LIN {X 0,Y 300.537,Z 1135.109,A -85,B 0,C 180,E1 14462.884,E2 14462.884} C_VEL
LIN {X 0,Y 304.265,Z 1129.427,A -85,B 0,C 180,E1 14457.835,E2 14457.835} C_VEL
LIN {X 0,Y 309.402,Z 1122.153,A -85,B 0,C 180,E1 14453.053,E2 14453.053} C_VEL
LIN {X 0,Y 314.973,Z 1114.845,A -85,B 0,C 180,E1 14449.161,E2 14449.161} C_VEL
LIN {X 0,Y 322.841,Z 1104.94,A -85,B 0,C 180,E1 14444.828,E2 14444.828} C_VEL
LIN {X 0,Y 331.827,Z 1093.472,A -85,B 0,C 180,E1 14440.835,E2 14440.835} C_VEL
LIN {X 0,Y 340.361,Z 1082.576,A -85,B 0,C 180,E1 14437.666,E2 14437.666} C_VEL
LIN {X 0,Y 350.994,Z 1068.769,A -85,B 0,C 180,E1 14434.299,E2 14434.299} C_VEL
LIN {X 0,Y 362.344,Z 1053.189,A -85,B 0,C 180,E1 14431.194,E2 14431.194} C_VEL
LIN {X 0,Y 369.861,Z 1042.527,A -85,B 0,C 180,E1 14429.373,E2 14429.373} C_VEL
LIN {X 0,Y 372.476,Z 1037.928,A -85,B 0,C 180,E1 14428.507,E2 14428.507} C_VEL
LIN {X 0,Y 377.031,Z 1026.802,A -85,B 0,C 180,E1 14426.039,E2 14426.039} C_VEL
LIN {X 0,Y 379.887,Z 1021.809,A -85,B 0,C 180,E1 14425.24,E2 14425.24} C_VEL
LIN {X 0,Y 392.376,Z 1001.673,A -85,B 0,C 180,E1 14422.92,E2 14422.92} C_VEL
LIN {X 0,Y 402.293,Z 984.331,A -85,B 0,C 180,E1 14421.248,E2 14421.248} C_VEL
LIN {X 0,Y 411.726,Z 966.45,A -85,B 0,C 180,E1 14419.775,E2 14419.775} C_VEL
LIN {X 0,Y 422.966,Z 942.726,A -85,B 0,C 180,E1 14418.141,E2 14418.141} C_VEL
LIN {X 0,Y 431.437,Z 922.389,A -85,B 0,C 180,E1 14416.979,E2 14416.979} C_VEL
LIN {X 0,Y 438.973,Z 902.071,A -85,B 0,C 180,E1 14415.999,E2 14415.999} C_VEL
LIN {X 0,Y 446.899,Z 877.548,A -85,B 0,C 180,E1 14415.019,E2 14415.019} C_VEL
LIN {X 0,Y 453.336,Z 852.946,A -85,B 0,C 180,E1 14414.24,E2 14414.24} C_VEL
LIN {X 0,Y 457.711,Z 832.707,A -85,B 0,C 180,E1 14413.717,E2 14413.717} C_VEL
LIN {X 0,Y 461.683,Z 809.62,A -85,B 0,C 180,E1 14413.245,E2 14413.245} C_VEL
LIN {X 0,Y 465.62,Z 774.989,A -85,B 0,C 180,E1 14412.698,E2 14412.698} C_VEL
LIN {X 0,Y 486.7,Z 556.586,A -85,B 0,C 180,E1 14409.493,E2 14409.493} C_VEL
LIN {X 0,Y 483.697,Z 550.634,A -85,B 0,C 180,E1 14407.185,E2 14407.185} C_VEL
LIN {X 0,Y 481.77,Z 547.068,A -85,B 0,C 180,E1 14405.359,E2 14405.359} C_VEL
LIN {X 0,Y 479.853,Z 543.385,A -85,B 0,C 180,E1 14402.867,E2 14402.867} C_VEL
LIN {X 0,Y 478.312,Z 540.425,A -85,B 0,C 180,E1 14398.443,E2 14398.443} C_VEL
LIN {X 0,Y 478.408,Z 540.862,A -85,B 0,C 180,E1 14396.285,E2 14396.285} C_VEL
LIN {X 0,Y 480.24,Z 544.178,A -85,B 0,C 180,E1 14392.162,E2 14392.162} C_VEL
LIN {X 0,Y 482.636,Z 548.887,A -85,B 0,C 180,E1 14389.375,E2 14389.375} C_VEL
LIN {X 0,Y 485.723,Z 554.856,A -85,B 0,C 180,E1 14386.822,E2 14386.822} C_VEL
LIN {X 0,Y 487.472,Z 558.564,A -85,B 0,C 180,E1 14385.592,E2 14385.592} C_VEL
LIN {X 0,Y 466.374,Z 778.807,A -85,B 0,C 180,E1 14382.251,E2 14382.251} C_VEL
LIN {X 0,Y 462.156,Z 819.105,A -85,B 0,C 180,E1 14381.613,E2 14381.613} C_VEL
LIN {X 0,Y 457.701,Z 845.254,A -85,B 0,C 180,E1 14381.12,E2 14381.12} C_VEL
LIN {X 0,Y 452.901,Z 867.044,A -85,B 0,C 180,E1 14380.637,E2 14380.637} C_VEL
LIN {X 0,Y 446.872,Z 889.838,A -85,B 0,C 180,E1 14380.007,E2 14380.007} C_VEL
LIN {X 0,Y 438.226,Z 917.079,A -85,B 0,C 180,E1 14379.046,E2 14379.046} C_VEL
LIN {X 0,Y 430.44,Z 938.212,A -85,B 0,C 180,E1 14378.123,E2 14378.123} C_VEL
LIN {X 0,Y 422.65,Z 957.244,A -85,B 0,C 180,E1 14377.137,E2 14377.137} C_VEL
LIN {X 0,Y 413.874,Z 976.767,A -85,B 0,C 180,E1 14375.95,E2 14375.95} C_VEL
LIN {X 0,Y 402.017,Z 1000.765,A -85,B 0,C 180,E1 14374.202,E2 14374.202} C_VEL
LIN {X 0,Y 390.581,Z 1021.665,A -85,B 0,C 180,E1 14372.342,E2 14372.342} C_VEL
LIN {X 0,Y 380.886,Z 1038.311,A -85,B 0,C 180,E1 14370.6,E2 14370.6} C_VEL
LIN {X 0,Y 370.782,Z 1054.723,A -85,B 0,C 180,E1 14368.607,E2 14368.607} C_VEL
LIN {X 0,Y 358.615,Z 1073.631,A -85,B 0,C 180,E1 14365.901,E2 14365.901} C_VEL
LIN {X 0,Y 346.466,Z 1091.434,A -85,B 0,C 180,E1 14362.797,E2 14362.797} C_VEL
LIN {X 0,Y 336.904,Z 1105.17,A -85,B 0,C 180,E1 14359.968,E2 14359.968} C_VEL
LIN {X 0,Y 327.706,Z 1118.263,A -85,B 0,C 180,E1 14356.82,E2 14356.82} C_VEL
LIN {X 0,Y 317.452,Z 1133.02,A -85,B 0,C 180,E1 14352.623,E2 14352.623} C_VEL
LIN {X 0,Y 308.488,Z 1146.151,A -85,B 0,C 180,E1 14348.012,E2 14348.012} C_VEL
LIN {X 0,Y 302.311,Z 1155.803,A -85,B 0,C 180,E1 14343.983,E2 14343.983} C_VEL
LIN {X 0,Y 297.196,Z 1164.602,A -85,B 0,C 180,E1 14339.64,E2 14339.64} C_VEL
LIN {X 0,Y 292.558,Z 1173.912,A -85,B 0,C 180,E1 14333.998,E2 14333.998} C_VEL
LIN {X 0,Y 290.123,Z 1180.103,A -85,B 0,C 180,E1 14329.208,E2 14329.208} C_VEL
LIN {X 0,Y 288.961,Z 1184.384,A -85,B 0,C 180,E1 14325.041,E2 14325.041} C_VEL
LIN {X 0,Y 288.442,Z 1187.555,A -85,B 0,C 180,E1 14320.991,E2 14320.991} C_VEL
LIN {X 0,Y 288.367,Z 1189.644,A -85,B 0,C 180,E1 14317.171,E2 14317.171} C_VEL
LIN {X 0,Y 288.427,Z 1190.814,A -85,B 0,C 180,E1 14313.379,E2 14313.379} C_VEL
LIN {X 0,Y 288.471,Z 1191.053,A -85,B 0,C 180,E1 14309.603,E2 14309.603} C_VEL
LIN {X 0,Y 288.431,Z 1190.344,A -85,B 0,C 180,E1 14305.825,E2 14305.825} C_VEL
LIN {X 0,Y 288.4,Z 1188.559,A -85,B 0,C 180,E1 14301.828,E2 14301.828} C_VEL
LIN {X 0,Y 288.599,Z 1185.626,A -85,B 0,C 180,E1 14297.697,E2 14297.697} C_VEL
LIN {X 0,Y 289.271,Z 1181.807,A -85,B 0,C 180,E1 14293.742,E2 14293.742} C_VEL
LIN {X 0,Y 290.606,Z 1176.811,A -85,B 0,C 180,E1 14289.666,E2 14289.666} C_VEL
LIN {X 0,Y 292.787,Z 1170.706,A -85,B 0,C 180,E1 14285.593,E2 14285.593} C_VEL
LIN {X 0,Y 295.918,Z 1163.458,A -85,B 0,C 180,E1 14281.549,E2 14281.549} C_VEL
LIN {X 0,Y 301.052,Z 1153.247,A -85,B 0,C 180,E1 14276.77,E2 14276.77} C_VEL
LIN {X 0,Y 307.763,Z 1141.001,A -85,B 0,C 180,E1 14272.119,E2 14272.119} C_VEL
LIN {X 0,Y 314.195,Z 1129.927,A -85,B 0,C 180,E1 14268.554,E2 14268.554} C_VEL
LIN {X 0,Y 321.498,Z 1117.681,A -85,B 0,C 180,E1 14265.162,E2 14265.162} C_VEL
LIN {X 0,Y 331.215,Z 1101.671,A -85,B 0,C 180,E1 14261.386,E2 14261.386} C_VEL
LIN {X 0,Y 341.43,Z 1084.347,A -85,B 0,C 180,E1 14258.024,E2 14258.024} C_VEL
LIN {X 0,Y 350.126,Z 1069.288,A -85,B 0,C 180,E1 14255.524,E2 14255.524} C_VEL
LIN {X 0,Y 359.111,Z 1053.183,A -85,B 0,C 180,E1 14253.21,E2 14253.21} C_VEL
LIN {X 0,Y 370.02,Z 1032.783,A -85,B 0,C 180,E1 14250.712,E2 14250.712} C_VEL
LIN {X 0,Y 380.326,Z 1011.808,A -85,B 0,C 180,E1 14248.587,E2 14248.587} C_VEL
LIN {X 0,Y 388.737,Z 993.522,A -85,B 0,C 180,E1 14246.999,E2 14246.999} C_VEL
LIN {X 0,Y 396.864,Z 974.565,A -85,B 0,C 180,E1 14245.586,E2 14245.586} C_VEL
LIN {X 0,Y 406.006,Z 951.26,A -85,B 0,C 180,E1 14244.107,E2 14244.107} C_VEL
LIN {X 0,Y 414.426,Z 926.626,A -85,B 0,C 180,E1 14242.835,E2 14242.835} C_VEL
LIN {X 0,Y 420.697,Z 905.998,A -85,B 0,C 180,E1 14241.953,E2 14241.953} C_VEL
LIN {X 0,Y 426.292,Z 884.993,A -85,B 0,C 180,E1 14241.2,E2 14241.2} C_VEL
LIN {X 0,Y 432.216,Z 858.983,A -85,B 0,C 180,E1 14240.452,E2 14240.452} C_VEL
LIN {X 0,Y 436.823,Z 831.955,A -85,B 0,C 180,E1 14239.859,E2 14239.859} C_VEL
LIN {X 0,Y 439.519,Z 809.536,A -85,B 0,C 180,E1 14239.442,E2 14239.442} C_VEL
LIN {X 0,Y 456.799,Z 596.987,A -85,B 0,C 180,E1 14236.09,E2 14236.09} C_VEL
LIN {X 0,Y 461.245,Z 542.225,A -85,B 0,C 180,E1 14235.207,E2 14235.207} C_VEL
LIN {X 0,Y 455.004,Z 530.522,A -85,B 0,C 180,E1 14232.598,E2 14232.598} C_VEL
LIN {X 0,Y 449.602,Z 520.756,A -85,B 0,C 180,E1 14229.99,E2 14229.99} C_VEL
LIN {X 0,Y 444.95,Z 512.775,A -85,B 0,C 180,E1 14227.359,E2 14227.359} C_VEL
LIN {X 0,Y 441.664,Z 507.167,A -85,B 0,C 180,E1 14225.131,E2 14225.131} C_VEL
LIN {X 0,Y 438.229,Z 501.32,A -85,B 0,C 180,E1 14222.223,E2 14222.223} C_VEL
LIN {X 0,Y 435.396,Z 496.62,A -85,B 0,C 180,E1 14218.816,E2 14218.816} C_VEL
LIN {X 0,Y 433.481,Z 493.881,A -85,B 0,C 180,E1 14213.909,E2 14213.909} C_VEL
LIN {X 0,Y 433.569,Z 494.107,A -85,B 0,C 180,E1 14211.111,E2 14211.111} C_VEL
LIN {X 0,Y 435.686,Z 496.998,A -85,B 0,C 180,E1 14206.394,E2 14206.394} C_VEL
LIN {X 0,Y 438.693,Z 502.126,A -85,B 0,C 180,E1 14202.969,E2 14202.969} C_VEL
LIN {X 0,Y 442.524,Z 508.361,A -85,B 0,C 180,E1 14199.913,E2 14199.913} C_VEL
LIN {X 0,Y 446.976,Z 516.099,A -85,B 0,C 180,E1 14197.093,E2 14197.093} C_VEL
LIN {X 0,Y 451.772,Z 524.554,A -85,B 0,C 180,E1 14194.572,E2 14194.572} C_VEL
LIN {X 0,Y 457.944,Z 536.068,A -85,B 0,C 180,E1 14191.789,E2 14191.789} C_VEL
LIN {X 0,Y 458.382,Z 537.284,A -85,B 0,C 180,E1 14191.59,E2 14191.59} C_VEL
LIN {X 0,Y 439.079,Z 769.572,A -85,B 0,C 180,E1 14188.029,E2 14188.029} C_VEL
LIN {X 0,Y 435.642,Z 805.367,A -85,B 0,C 180,E1 14187.439,E2 14187.439} C_VEL
LIN {X 0,Y 431.934,Z 829.629,A -85,B 0,C 180,E1 14186.906,E2 14186.906} C_VEL
LIN {X 0,Y 427.887,Z 850.615,A -85,B 0,C 180,E1 14186.314,E2 14186.314} C_VEL
LIN {X 0,Y 422.274,Z 874.564,A -85,B 0,C 180,E1 14185.486,E2 14185.486} C_VEL
LIN {X 0,Y 415.381,Z 898.542,A -85,B 0,C 180,E1 14184.448,E2 14184.448} C_VEL
LIN {X 0,Y 408.612,Z 919.046,A -85,B 0,C 180,E1 14183.379,E2 14183.379} C_VEL
LIN {X 0,Y 400.988,Z 939.639,A -85,B 0,C 180,E1 14182.11,E2 14182.11} C_VEL
LIN {X 0,Y 390.967,Z 963.549,A -85,B 0,C 180,E1 14180.334,E2 14180.334} C_VEL
LIN {X 0,Y 382.521,Z 981.74,A -85,B 0,C 180,E1 14178.719,E2 14178.719} C_VEL
LIN {X 0,Y 374.05,Z 998.65,A -85,B 0,C 180,E1 14176.977,E2 14176.977} C_VEL
LIN {X 0,Y 363.351,Z 1018.538,A -85,B 0,C 180,E1 14174.563,E2 14174.563} C_VEL
LIN {X 0,Y 352.953,Z 1036.284,A -85,B 0,C 180,E1 14171.955,E2 14171.955} C_VEL
LIN {X 0,Y 344.235,Z 1050.501,A -85,B 0,C 180,E1 14169.502,E2 14169.502} C_VEL
LIN {X 0,Y 334.277,Z 1066.205,A -85,B 0,C 180,E1 14166.316,E2 14166.316} C_VEL
LIN {X 0,Y 324.82,Z 1080.383,A -85,B 0,C 180,E1 14162.803,E2 14162.803} C_VEL
LIN {X 0,Y 317.181,Z 1091.77,A -85,B 0,C 180,E1 14159.456,E2 14159.456} C_VEL
LIN {X 0,Y 309.26,Z 1103.755,A -85,B 0,C 180,E1 14155.262,E2 14155.262} C_VEL
LIN {X 0,Y 302.465,Z 1114.131,A -85,B 0,C 180,E1 14150.714,E2 14150.714} C_VEL
LIN {X 0,Y 297.915,Z 1121.561,A -85,B 0,C 180,E1 14146.776,E2 14146.776} C_VEL
LIN {X 0,Y 293.861,Z 1128.975,A -85,B 0,C 180,E1 14141.979,E2 14141.979} C_VEL
LIN {X 0,Y 291.048,Z 1134.872,A -85,B 0,C 180,E1 14136.906,E2 14136.906} C_VEL
LIN {X 0,Y 289.685,Z 1138.521,A -85,B 0,C 180,E1 14132.77,E2 14132.77} C_VEL
LIN {X 0,Y 289.008,Z 1141.071,A -85,B 0,C 180,E1 14128.81,E2 14128.81} C_VEL
LIN {X 0,Y 288.706,Z 1142.744,A -85,B 0,C 180,E1 14124.834,E2 14124.834} C_VEL
LIN {X 0,Y 288.659,Z 1143.577,A -85,B 0,C 180,E1 14120.63,E2 14120.63} C_VEL
LIN {X 0,Y 288.869,Z 1143.374,A -85,B 0,C 180,E1 14115.742,E2 14115.742} C_VEL
LIN {X 0,Y 289.497,Z 1141.838,A -85,B 0,C 180,E1 14111.055,E2 14111.055} C_VEL
LIN {X 0,Y 290.733,Z 1139.376,A -85,B 0,C 180,E1 14106.703,E2 14106.703} C_VEL
LIN {X 0,Y 292.756,Z 1136.021,A -85,B 0,C 180,E1 14102.544,E2 14102.544} C_VEL
LIN {X 0,Y 296.29,Z 1130.917,A -85,B 0,C 180,E1 14097.779,E2 14097.779} C_VEL
LIN {X 0,Y 301.799,Z 1123.582,A -85,B 0,C 180,E1 14092.669,E2 14092.669} C_VEL
LIN {X 0,Y 307.578,Z 1116.356,A -85,B 0,C 180,E1 14088.673,E2 14088.673} C_VEL
LIN {X 0,Y 314.486,Z 1107.977,A -85,B 0,C 180,E1 14084.847,E2 14084.847} C_VEL
LIN {X 0,Y 324.399,Z 1096.058,A -85,B 0,C 180,E1 14080.421,E2 14080.421} C_VEL
LIN {X 0,Y 333.918,Z 1084.361,A -85,B 0,C 180,E1 14076.919,E2 14076.919} C_VEL
LIN {X 0,Y 343.428,Z 1072.444,A -85,B 0,C 180,E1 14073.927,E2 14073.927} C_VEL
LIN {X 0,Y 354.974,Z 1057.507,A -85,B 0,C 180,E1 14070.785,E2 14070.785} C_VEL
LIN {X 0,Y 366.845,Z 1040.993,A -85,B 0,C 180,E1 14067.957,E2 14067.957} C_VEL
LIN {X 0,Y 376.707,Z 1026.562,A -85,B 0,C 180,E1 14065.871,E2 14065.871} C_VEL
LIN {X 0,Y 379.887,Z 1021.809,A -85,B 0,C 180,E1 14065.24,E2 14065.24} C_VEL
LIN {X 0,Y 382.759,Z 1016.786,A -85,B 0,C 180,E1 14064.46,E2 14064.46} C_VEL
LIN {X 0,Y 387.816,Z 1004.51,A -85,B 0,C 180,E1 14062.214,E2 14062.214} C_VEL
LIN {X 0,Y 390.69,Z 999.056,A -85,B 0,C 180,E1 14061.518,E2 14061.518} C_VEL
LIN {X 0,Y 402,Z 979.461,A -85,B 0,C 180,E1 14059.711,E2 14059.711} C_VEL
LIN {X 0,Y 413.33,Z 957.464,A -85,B 0,C 180,E1 14058.038,E2 14058.038} C_VEL
LIN {X 0,Y 422.043,Z 938.688,A -85,B 0,C 180,E1 14056.841,E2 14056.841} C_VEL
LIN {X 0,Y 429.75,Z 920.272,A -85,B 0,C 180,E1 14055.835,E2 14055.835} C_VEL
LIN {X 0,Y 438.408,Z 896.971,A -85,B 0,C 180,E1 14054.761,E2 14054.761} C_VEL
LIN {X 0,Y 446.121,Z 871.943,A -85,B 0,C 180,E1 14053.83,E2 14053.83} C_VEL
LIN {X 0,Y 451.666,Z 850.593,A -85,B 0,C 180,E1 14053.189,E2 14053.189} C_VEL
LIN {X 0,Y 456.216,Z 829.368,A -85,B 0,C 180,E1 14052.672,E2 14052.672} C_VEL
LIN {X 0,Y 460.774,Z 800.806,A -85,B 0,C 180,E1 14052.134,E2 14052.134} C_VEL
LIN {X 0,Y 467.223,Z 736.827,A -85,B 0,C 180,E1 14051.18,E2 14051.18} C_VEL
LIN {X 0,Y 484.477,Z 562.449,A -85,B 0,C 180,E1 14048.638,E2 14048.638} C_VEL
LIN {X 0,Y 481.658,Z 556.855,A -85,B 0,C 180,E1 14046.257,E2 14046.257} C_VEL
LIN {X 0,Y 480.236,Z 554.244,A -85,B 0,C 180,E1 14044.777,E2 14044.777} C_VEL
LIN {X 0,Y 478.793,Z 551.264,A -85,B 0,C 180,E1 14042.753,E2 14042.753} C_VEL
LIN {X 0,Y 477.333,Z 548.368,A -85,B 0,C 180,E1 14038.44,E2 14038.44} C_VEL
LIN {X 0,Y 477.428,Z 548.825,A -85,B 0,C 180,E1 14036.277,E2 14036.277} C_VEL
LIN {X 0,Y 479.17,Z 552.085,A -85,B 0,C 180,E1 14032.265,E2 14032.265} C_VEL
LIN {X 0,Y 481.458,Z 556.712,A -85,B 0,C 180,E1 14029.53,E2 14029.53} C_VEL
LIN {X 0,Y 484.362,Z 562.5,A -85,B 0,C 180,E1 14027.057,E2 14027.057} C_VEL
LIN {X 0,Y 485.184,Z 564.508,A -85,B 0,C 180,E1 14026.429,E2 14026.429} C_VEL
LIN {X 0,Y 463.683,Z 784.434,A -85,B 0,C 180,E1 14023.119,E2 14023.119} C_VEL
LIN {X 0,Y 459.613,Z 820.838,A -85,B 0,C 180,E1 14022.54,E2 14022.54} C_VEL
LIN {X 0,Y 455.315,Z 845.433,A -85,B 0,C 180,E1 14022.08,E2 14022.08} C_VEL
LIN {X 0,Y 450.433,Z 867.156,A -85,B 0,C 180,E1 14021.606,E2 14021.606} C_VEL
LIN {X 0,Y 444.198,Z 890.257,A -85,B 0,C 180,E1 14020.978,E2 14020.978} C_VEL
LIN {X 0,Y 435.57,Z 916.837,A -85,B 0,C 180,E1 14020.054,E2 14020.054} C_VEL
LIN {X 0,Y 427.491,Z 938.335,A -85,B 0,C 180,E1 14019.13,E2 14019.13} C_VEL
LIN {X 0,Y 419.166,Z 958.203,A -85,B 0,C 180,E1 14018.11,E2 14018.11} C_VEL
LIN {X 0,Y 408.705,Z 980.824,A -85,B 0,C 180,E1 14016.726,E2 14016.726} C_VEL
LIN {X 0,Y 396.643,Z 1004.01,A -85,B 0,C 180,E1 14014.989,E2 14014.989} C_VEL
LIN {X 0,Y 386.093,Z 1022.735,A -85,B 0,C 180,E1 14013.309,E2 14013.309} C_VEL
LIN {X 0,Y 375.577,Z 1040.217,A -85,B 0,C 180,E1 14011.465,E2 14011.465} C_VEL
LIN {X 0,Y 362.21,Z 1061.073,A -85,B 0,C 180,E1 14008.841,E2 14008.841} C_VEL
LIN {X 0,Y 350.273,Z 1078.53,A -85,B 0,C 180,E1 14006.167,E2 14006.167} C_VEL
LIN {X 0,Y 340.082,Z 1092.943,A -85,B 0,C 180,E1 14003.565,E2 14003.565} C_VEL
LIN {X 0,Y 329.944,Z 1106.956,A -85,B 0,C 180,E1 14000.601,E2 14000.601} C_VEL
LIN {X 0,Y 318.077,Z 1123.167,A -85,B 0,C 180,E1 13996.493,E2 13996.493} C_VEL
LIN {X 0,Y 308.439,Z 1136.343,A -85,B 0,C 180,E1 13992.397,E2 13992.397} C_VEL
LIN {X 0,Y 300.832,Z 1147.106,A -85,B 0,C 180,E1 13988.427,E2 13988.427} C_VEL
LIN {X 0,Y 293.717,Z 1157.873,A -85,B 0,C 180,E1 13983.702,E2 13983.702} C_VEL
LIN {X 0,Y 287.693,Z 1167.93,A -85,B 0,C 180,E1 13978.207,E2 13978.207} C_VEL
LIN {X 0,Y 284.27,Z 1174.726,A -85,B 0,C 180,E1 13973.639,E2 13973.639} C_VEL
LIN {X 0,Y 282.194,Z 1179.841,A -85,B 0,C 180,E1 13969.455,E2 13969.455} C_VEL
LIN {X 0,Y 281.004,Z 1183.953,A -85,B 0,C 180,E1 13965.266,E2 13965.266} C_VEL
LIN {X 0,Y 280.458,Z 1187.061,A -85,B 0,C 180,E1 13961.1,E2 13961.1} C_VEL
LIN {X 0,Y 280.386,Z 1189.088,A -85,B 0,C 180,E1 13957.17,E2 13957.17} C_VEL
LIN {X 0,Y 280.448,Z 1190.164,A -85,B 0,C 180,E1 13953.475,E2 13953.475} C_VEL
LIN {X 0,Y 280.502,Z 1190.406,A -85,B 0,C 180,E1 13949.796,E2 13949.796} C_VEL
LIN {X 0,Y 280.458,Z 1189.728,A -85,B 0,C 180,E1 13945.911,E2 13945.911} C_VEL
LIN {X 0,Y 280.421,Z 1187.969,A -85,B 0,C 180,E1 13941.801,E2 13941.801} C_VEL
LIN {X 0,Y 280.632,Z 1185.008,A -85,B 0,C 180,E1 13937.492,E2 13937.492} C_VEL
LIN {X 0,Y 281.381,Z 1181.029,A -85,B 0,C 180,E1 13933.272,E2 13933.272} C_VEL
LIN {X 0,Y 282.844,Z 1176.003,A -85,B 0,C 180,E1 13929.082,E2 13929.082} C_VEL
LIN {X 0,Y 285.176,Z 1169.864,A -85,B 0,C 180,E1 13924.898,E2 13924.898} C_VEL
LIN {X 0,Y 288.723,Z 1162.189,A -85,B 0,C 180,E1 13920.544,E2 13920.544} C_VEL
LIN {X 0,Y 294.766,Z 1150.85,A -85,B 0,C 180,E1 13915.26,E2 13915.26} C_VEL
LIN {X 0,Y 301.381,Z 1139.443,A -85,B 0,C 180,E1 13910.925,E2 13910.925} C_VEL
LIN {X 0,Y 308.194,Z 1128.259,A -85,B 0,C 180,E1 13907.309,E2 13907.309} C_VEL
LIN {X 0,Y 317.016,Z 1114.199,A -85,B 0,C 180,E1 13903.44,E2 13903.44} C_VEL
LIN {X 0,Y 327.315,Z 1097.626,A -85,B 0,C 180,E1 13899.665,E2 13899.665} C_VEL
LIN {X 0,Y 336.47,Z 1082.641,A -85,B 0,C 180,E1 13896.789,E2 13896.789} C_VEL
LIN {X 0,Y 345.496,Z 1067.483,A -85,B 0,C 180,E1 13894.287,E2 13894.287} C_VEL
LIN {X 0,Y 356.049,Z 1049.098,A -85,B 0,C 180,E1 13891.692,E2 13891.692} C_VEL
LIN {X 0,Y 367.58,Z 1027.575,A -85,B 0,C 180,E1 13889.173,E2 13889.173} C_VEL
LIN {X 0,Y 376.657,Z 1009.479,A -85,B 0,C 180,E1 13887.384,E2 13887.384} C_VEL
LIN {X 0,Y 385.36,Z 990.871,A -85,B 0,C 180,E1 13885.799,E2 13885.799} C_VEL
LIN {X 0,Y 395.465,Z 967.525,A -85,B 0,C 180,E1 13884.116,E2 13884.116} C_VEL
LIN {X 0,Y 404.378,Z 944.142,A -85,B 0,C 180,E1 13882.74,E2 13882.74} C_VEL
LIN {X 0,Y 411.228,Z 924.212,A -85,B 0,C 180,E1 13881.753,E2 13881.753} C_VEL
LIN {X 0,Y 417.625,Z 903.327,A -85,B 0,C 180,E1 13880.882,E2 13880.882} C_VEL
LIN {X 0,Y 424.134,Z 878.897,A -85,B 0,C 180,E1 13880.045,E2 13880.045} C_VEL
LIN {X 0,Y 429.959,Z 851.7,A -85,B 0,C 180,E1 13879.329,E2 13879.329} C_VEL
LIN {X 0,Y 433.712,Z 829.135,A -85,B 0,C 180,E1 13878.854,E2 13878.854} C_VEL
LIN {X 0,Y 436.465,Z 805.631,A -85,B 0,C 180,E1 13878.427,E2 13878.427} C_VEL
LIN {X 0,Y 454.775,Z 585.097,A -85,B 0,C 180,E1 13874.969,E2 13874.969} C_VEL
LIN {X 0,Y 457.922,Z 547.005,A -85,B 0,C 180,E1 13874.349,E2 13874.349} C_VEL
LIN {X 0,Y 451.436,Z 534.659,A -85,B 0,C 180,E1 13871.466,E2 13871.466} C_VEL
LIN {X 0,Y 446.147,Z 524.973,A -85,B 0,C 180,E1 13868.701,E2 13868.701} C_VEL
LIN {X 0,Y 441.264,Z 516.386,A -85,B 0,C 180,E1 13865.592,E2 13865.592} C_VEL
LIN {X 0,Y 438.176,Z 511.224,A -85,B 0,C 180,E1 13863.139,E2 13863.139} C_VEL
LIN {X 0,Y 436.559,Z 508.515,A -85,B 0,C 180,E1 13861.575,E2 13861.575} C_VEL
LIN {X 0,Y 434.317,Z 504.493,A -85,B 0,C 180,E1 13858.681,E2 13858.681} C_VEL
LIN {X 0,Y 432.488,Z 501.79,A -85,B 0,C 180,E1 13853.762,E2 13853.762} C_VEL
LIN {X 0,Y 432.641,Z 502.177,A -85,B 0,C 180,E1 13850.824,E2 13850.824} C_VEL
LIN {X 0,Y 434.621,Z 504.931,A -85,B 0,C 180,E1 13846.496,E2 13846.496} C_VEL
LIN {X 0,Y 437.445,Z 509.843,A -85,B 0,C 180,E1 13843.193,E2 13843.193} C_VEL
LIN {X 0,Y 441.189,Z 516.081,A -85,B 0,C 180,E1 13840.126,E2 13840.126} C_VEL
LIN {X 0,Y 446.122,Z 524.774,A -85,B 0,C 180,E1 13836.977,E2 13836.977} C_VEL
LIN {X 0,Y 451.434,Z 534.583,A -85,B 0,C 180,E1 13834.2,E2 13834.2} C_VEL
LIN {X 0,Y 455.197,Z 542.032,A -85,B 0,C 180,E1 13832.463,E2 13832.463} C_VEL
LIN {X 0,Y 435.378,Z 775.307,A -85,B 0,C 180,E1 13828.902,E2 13828.902} C_VEL
LIN {X 0,Y 431.882,Z 808.711,A -85,B 0,C 180,E1 13828.339,E2 13828.339} C_VEL
LIN {X 0,Y 428.305,Z 831.266,A -85,B 0,C 180,E1 13827.84,E2 13827.84} C_VEL
LIN {X 0,Y 423.962,Z 853.086,A -85,B 0,C 180,E1 13827.22,E2 13827.22} C_VEL
LIN {X 0,Y 417.6,Z 878.875,A -85,B 0,C 180,E1 13826.306,E2 13826.306} C_VEL
LIN {X 0,Y 411.208,Z 900.34,A -85,B 0,C 180,E1 13825.366,E2 13825.366} C_VEL
LIN {X 0,Y 404.382,Z 920.504,A -85,B 0,C 180,E1 13824.315,E2 13824.315} C_VEL
LIN {X 0,Y 395.606,Z 943.583,A -85,B 0,C 180,E1 13822.882,E2 13822.882} C_VEL
LIN {X 0,Y 386.037,Z 965.466,A -85,B 0,C 180,E1 13821.224,E2 13821.224} C_VEL
LIN {X 0,Y 377.731,Z 982.894,A -85,B 0,C 180,E1 13819.671,E2 13819.671} C_VEL
LIN {X 0,Y 368.756,Z 1000.33,A -85,B 0,C 180,E1 13817.866,E2 13817.866} C_VEL
LIN {X 0,Y 357.214,Z 1021.004,A -85,B 0,C 180,E1 13815.313,E2 13815.313} C_VEL
LIN {X 0,Y 347.684,Z 1036.837,A -85,B 0,C 180,E1 13812.965,E2 13812.965} C_VEL
LIN {X 0,Y 338.696,Z 1051.059,A -85,B 0,C 180,E1 13810.5,E2 13810.5} C_VEL
LIN {X 0,Y 328.407,Z 1066.77,A -85,B 0,C 180,E1 13807.291,E2 13807.291} C_VEL
LIN {X 0,Y 318.507,Z 1081.105,A -85,B 0,C 180,E1 13803.703,E2 13803.703} C_VEL
LIN {X 0,Y 310.663,Z 1092.36,A -85,B 0,C 180,E1 13800.351,E2 13800.351} C_VEL
LIN {X 0,Y 302.407,Z 1104.35,A -85,B 0,C 180,E1 13796.087,E2 13796.087} C_VEL
LIN {X 0,Y 295.287,Z 1114.736,A -85,B 0,C 180,E1 13791.45,E2 13791.45} C_VEL
LIN {X 0,Y 290.504,Z 1122.174,A -85,B 0,C 180,E1 13787.424,E2 13787.424} C_VEL
LIN {X 0,Y 286.36,Z 1129.311,A -85,B 0,C 180,E1 13782.707,E2 13782.707} C_VEL
LIN {X 0,Y 283.329,Z 1135.307,A -85,B 0,C 180,E1 13777.502,E2 13777.502} C_VEL
LIN {X 0,Y 281.845,Z 1139.002,A -85,B 0,C 180,E1 13773.254,E2 13773.254} C_VEL
LIN {X 0,Y 281.082,Z 1141.601,A -85,B 0,C 180,E1 13769.185,E2 13769.185} C_VEL
LIN {X 0,Y 280.742,Z 1143.322,A -85,B 0,C 180,E1 13765.096,E2 13765.096} C_VEL
LIN {X 0,Y 280.684,Z 1144.15,A -85,B 0,C 180,E1 13761.189,E2 13761.189} C_VEL
LIN {X 0,Y 280.801,Z 1144.191,A -85,B 0,C 180,E1 13757.246,E2 13757.246} C_VEL
LIN {X 0,Y 281.221,Z 1143.317,A -85,B 0,C 180,E1 13752.836,E2 13752.836} C_VEL
LIN {X 0,Y 282.489,Z 1140.929,A -85,B 0,C 180,E1 13747.493,E2 13747.493} C_VEL
LIN {X 0,Y 284.73,Z 1137.314,A -85,B 0,C 180,E1 13742.612,E2 13742.612} C_VEL
LIN {X 0,Y 287.941,Z 1132.843,A -85,B 0,C 180,E1 13738.142,E2 13738.142} C_VEL
LIN {X 0,Y 293.166,Z 1126.335,A -85,B 0,C 180,E1 13733.112,E2 13733.112} C_VEL
LIN {X 0,Y 300.115,Z 1117.979,A -85,B 0,C 180,E1 13728.216,E2 13728.216} C_VEL
LIN {X 0,Y 307.278,Z 1109.674,A -85,B 0,C 180,E1 13724.286,E2 13724.286} C_VEL
LIN {X 0,Y 316.107,Z 1099.547,A -85,B 0,C 180,E1 13720.333,E2 13720.333} C_VEL
LIN {X 0,Y 327.258,Z 1086.486,A -85,B 0,C 180,E1 13716.236,E2 13716.236} C_VEL
LIN {X 0,Y 337.002,Z 1074.731,A -85,B 0,C 180,E1 13713.21,E2 13713.21} C_VEL
LIN {X 0,Y 347.14,Z 1062.066,A -85,B 0,C 180,E1 13710.461,E2 13710.461} C_VEL
LIN {X 0,Y 359.718,Z 1045.606,A -85,B 0,C 180,E1 13707.479,E2 13707.479} C_VEL
LIN {X 0,Y 371.888,Z 1028.331,A -85,B 0,C 180,E1 13704.931,E2 13704.931} C_VEL
LIN {X 0,Y 381.926,Z 1013.186,A -85,B 0,C 180,E1 13703.044,E2 13703.044} C_VEL
LIN {X 0,Y 390.69,Z 999.056,A -85,B 0,C 180,E1 13701.518,E2 13701.518} C_VEL
LIN {X 0,Y 393.614,Z 993.646,A -85,B 0,C 180,E1 13700.837,E2 13700.837} C_VEL
LIN {X 0,Y 399.416,Z 979.519,A -85,B 0,C 180,E1 13698.7,E2 13698.7} C_VEL
LIN {X 0,Y 401.876,Z 974.446,A -85,B 0,C 180,E1 13698.193,E2 13698.193} C_VEL
LIN {X 0,Y 411.568,Z 955.661,A -85,B 0,C 180,E1 13696.828,E2 13696.828} C_VEL
LIN {X 0,Y 420.524,Z 936.504,A -85,B 0,C 180,E1 13695.646,E2 13695.646} C_VEL
LIN {X 0,Y 430.075,Z 913.662,A -85,B 0,C 180,E1 13694.465,E2 13694.465} C_VEL
LIN {X 0,Y 438.341,Z 890.26,A -85,B 0,C 180,E1 13693.478,E2 13693.478} C_VEL
LIN {X 0,Y 444.435,Z 870.294,A -85,B 0,C 180,E1 13692.772,E2 13692.772} C_VEL
LIN {X 0,Y 450.149,Z 848.259,A -85,B 0,C 180,E1 13692.133,E2 13692.133} C_VEL
LIN {X 0,Y 455.763,Z 820.838,A -85,B 0,C 180,E1 13691.516,E2 13691.516} C_VEL
LIN {X 0,Y 459.199,Z 797.378,A -85,B 0,C 180,E1 13691.11,E2 13691.11} C_VEL
LIN {X 0,Y 482.378,Z 568.599,A -85,B 0,C 180,E1 13687.803,E2 13687.803} C_VEL
LIN {X 0,Y 479.803,Z 563.168,A -85,B 0,C 180,E1 13685.381,E2 13685.381} C_VEL
LIN {X 0,Y 477.735,Z 559.143,A -85,B 0,C 180,E1 13682.639,E2 13682.639} C_VEL
LIN {X 0,Y 476.348,Z 556.281,A -85,B 0,C 180,E1 13678.316,E2 13678.316} C_VEL
LIN {X 0,Y 476.467,Z 556.865,A -85,B 0,C 180,E1 13676.149,E2 13676.149} C_VEL
LIN {X 0,Y 478.065,Z 559.891,A -85,B 0,C 180,E1 13672.428,E2 13672.428} C_VEL
LIN {X 0,Y 480.228,Z 564.407,A -85,B 0,C 180,E1 13669.745,E2 13669.745} C_VEL
LIN {X 0,Y 483.024,Z 570.178,A -85,B 0,C 180,E1 13667.281,E2 13667.281} C_VEL
LIN {X 0,Y 461.679,Z 784.151,A -85,B 0,C 180,E1 13664.085,E2 13664.085} C_VEL
LIN {X 0,Y 457.542,Z 820.416,A -85,B 0,C 180,E1 13663.515,E2 13663.515} C_VEL
LIN {X 0,Y 453.207,Z 844.884,A -85,B 0,C 180,E1 13663.065,E2 13663.065} C_VEL
LIN {X 0,Y 448.256,Z 866.638,A -85,B 0,C 180,E1 13662.601,E2 13662.601} C_VEL
LIN {X 0,Y 441.863,Z 889.971,A -85,B 0,C 180,E1 13661.981,E2 13661.981} C_VEL
LIN {X 0,Y 433.307,Z 915.938,A -85,B 0,C 180,E1 13661.099,E2 13661.099} C_VEL
LIN {X 0,Y 425.083,Z 937.466,A -85,B 0,C 180,E1 13660.196,E2 13660.196} C_VEL
LIN {X 0,Y 416.545,Z 957.495,A -85,B 0,C 180,E1 13659.19,E2 13659.19} C_VEL
LIN {X 0,Y 405.932,Z 980.014,A -85,B 0,C 180,E1 13657.84,E2 13657.84} C_VEL
LIN {X 0,Y 393.613,Z 1003.233,A -85,B 0,C 180,E1 13656.131,E2 13656.131} C_VEL
LIN {X 0,Y 383.188,Z 1021.349,A -85,B 0,C 180,E1 13654.532,E2 13654.532} C_VEL
LIN {X 0,Y 373.091,Z 1037.773,A -85,B 0,C 180,E1 13652.84,E2 13652.84} C_VEL
LIN {X 0,Y 361.978,Z 1054.801,A -85,B 0,C 180,E1 13650.792,E2 13650.792} C_VEL
LIN {X 0,Y 347.552,Z 1075.623,A -85,B 0,C 180,E1 13647.757,E2 13647.757} C_VEL
LIN {X 0,Y 336.521,Z 1090.733,A -85,B 0,C 180,E1 13645.089,E2 13645.089} C_VEL
LIN {X 0,Y 325.952,Z 1104.812,A -85,B 0,C 180,E1 13642.155,E2 13642.155} C_VEL
LIN {X 0,Y 315.345,Z 1118.751,A -85,B 0,C 180,E1 13638.716,E2 13638.716} C_VEL
LIN {X 0,Y 303.449,Z 1134.251,A -85,B 0,C 180,E1 13634.046,E2 13634.046} C_VEL
LIN {X 0,Y 295.282,Z 1145.157,A -85,B 0,C 180,E1 13630.043,E2 13630.043} C_VEL
LIN {X 0,Y 288.42,Z 1154.763,A -85,B 0,C 180,E1 13625.864,E2 13625.864} C_VEL
LIN {X 0,Y 282.209,Z 1164.276,A -85,B 0,C 180,E1 13620.913,E2 13620.913} C_VEL
LIN {X 0,Y 277.141,Z 1173.149,A -85,B 0,C 180,E1 13615.098,E2 13615.098} C_VEL
LIN {X 0,Y 274.579,Z 1178.786,A -85,B 0,C 180,E1 13610.462,E2 13610.462} C_VEL
LIN {X 0,Y 273.142,Z 1183.162,A -85,B 0,C 180,E1 13605.935,E2 13605.935} C_VEL
LIN {X 0,Y 272.503,Z 1186.307,A -85,B 0,C 180,E1 13601.643,E2 13601.643} C_VEL
LIN {X 0,Y 272.399,Z 1188.37,A -85,B 0,C 180,E1 13597.593,E2 13597.593} C_VEL
LIN {X 0,Y 272.464,Z 1189.481,A -85,B 0,C 180,E1 13593.788,E2 13593.788} C_VEL
LIN {X 0,Y 272.537,Z 1189.758,A -85,B 0,C 180,E1 13590,E2 13590} C_VEL
LIN {X 0,Y 272.485,Z 1189.109,A -85,B 0,C 180,E1 13586.002,E2 13586.002} C_VEL
LIN {X 0,Y 272.442,Z 1187.375,A -85,B 0,C 180,E1 13581.771,E2 13581.771} C_VEL
LIN {X 0,Y 272.665,Z 1184.39,A -85,B 0,C 180,E1 13577.279,E2 13577.279} C_VEL
LIN {X 0,Y 273.444,Z 1180.48,A -85,B 0,C 180,E1 13572.991,E2 13572.991} C_VEL
LIN {X 0,Y 275.098,Z 1175.191,A -85,B 0,C 180,E1 13568.464,E2 13568.464} C_VEL
LIN {X 0,Y 277.767,Z 1168.681,A -85,B 0,C 180,E1 13563.95,E2 13563.95} C_VEL
LIN {X 0,Y 282.481,Z 1159.358,A -85,B 0,C 180,E1 13558.647,E2 13558.647} C_VEL
LIN {X 0,Y 288.691,Z 1148.394,A -85,B 0,C 180,E1 13553.684,E2 13553.684} C_VEL
LIN {X 0,Y 294.78,Z 1138.437,A -85,B 0,C 180,E1 13549.875,E2 13549.875} C_VEL
LIN {X 0,Y 301.948,Z 1127.215,A -85,B 0,C 180,E1 13546.206,E2 13546.206} C_VEL
LIN {X 0,Y 311.66,Z 1112.397,A -85,B 0,C 180,E1 13542.108,E2 13542.108} C_VEL
LIN {X 0,Y 322.401,Z 1095.597,A -85,B 0,C 180,E1 13538.314,E2 13538.314} C_VEL
LIN {X 0,Y 331.663,Z 1080.929,A -85,B 0,C 180,E1 13535.515,E2 13535.515} C_VEL
LIN {X 0,Y 341.63,Z 1064.671,A -85,B 0,C 180,E1 13532.863,E2 13532.863} C_VEL
LIN {X 0,Y 354.175,Z 1043.059,A -85,B 0,C 180,E1 13529.925,E2 13529.925} C_VEL
LIN {X 0,Y 364.15,Z 1024.725,A -85,B 0,C 180,E1 13527.856,E2 13527.856} C_VEL
LIN {X 0,Y 373.16,Z 1007.113,A -85,B 0,C 180,E1 13526.155,E2 13526.155} C_VEL
LIN {X 0,Y 383.02,Z 986.396,A -85,B 0,C 180,E1 13524.441,E2 13524.441} C_VEL
LIN {X 0,Y 393.571,Z 961.704,A -85,B 0,C 180,E1 13522.752,E2 13522.752} C_VEL
LIN {X 0,Y 401.571,Z 940.874,A -85,B 0,C 180,E1 13521.571,E2 13521.571} C_VEL
LIN {X 0,Y 408.572,Z 920.593,A -85,B 0,C 180,E1 13520.601,E2 13520.601} C_VEL
LIN {X 0,Y 416.108,Z 895.916,A -85,B 0,C 180,E1 13519.623,E2 13519.623} C_VEL
LIN {X 0,Y 422.697,Z 869.575,A -85,B 0,C 180,E1 13518.807,E2 13518.807} C_VEL
LIN {X 0,Y 427.267,Z 847.596,A -85,B 0,C 180,E1 13518.271,E2 13518.271} C_VEL
LIN {X 0,Y 431.105,Z 823.745,A -85,B 0,C 180,E1 13517.785,E2 13517.785} C_VEL
LIN {X 0,Y 434.738,Z 787.74,A -85,B 0,C 180,E1 13517.178,E2 13517.178} C_VEL
LIN {X 0,Y 453.561,Z 565.817,A -85,B 0,C 180,E1 13513.724,E2 13513.724} C_VEL
LIN {X 0,Y 454.695,Z 551.854,A -85,B 0,C 180,E1 13513.48,E2 13513.48} C_VEL
LIN {X 0,Y 448.58,Z 540.001,A -85,B 0,C 180,E1 13510.603,E2 13510.603} C_VEL
LIN {X 0,Y 443.802,Z 531.208,A -85,B 0,C 180,E1 13507.965,E2 13507.965} C_VEL
LIN {X 0,Y 439.537,Z 523.483,A -85,B 0,C 180,E1 13505.09,E2 13505.09} C_VEL
LIN {X 0,Y 436.6,Z 518.368,A -85,B 0,C 180,E1 13502.625,E2 13502.625} C_VEL
LIN {X 0,Y 435.065,Z 515.86,A -85,B 0,C 180,E1 13501.054,E2 13501.054} C_VEL
LIN {X 0,Y 433.241,Z 512.366,A -85,B 0,C 180,E1 13498.545,E2 13498.545} C_VEL
LIN {X 0,Y 431.508,Z 509.729,A -85,B 0,C 180,E1 13493.743,E2 13493.743} C_VEL
LIN {X 0,Y 431.665,Z 510.136,A -85,B 0,C 180,E1 13490.803,E2 13490.803} C_VEL
LIN {X 0,Y 433.556,Z 512.864,A -85,B 0,C 180,E1 13486.598,E2 13486.598} C_VEL
LIN {X 0,Y 436.303,Z 517.764,A -85,B 0,C 180,E1 13483.317,E2 13483.317} C_VEL
LIN {X 0,Y 439.951,Z 523.942,A -85,B 0,C 180,E1 13480.275,E2 13480.275} C_VEL
LIN {X 0,Y 444.684,Z 532.591,A -85,B 0,C 180,E1 13477.185,E2 13477.185} C_VEL
LIN {X 0,Y 449.635,Z 541.967,A -85,B 0,C 180,E1 13474.532,E2 13474.532} C_VEL
LIN {X 0,Y 452.095,Z 547.044,A -85,B 0,C 180,E1 13473.344,E2 13473.344} C_VEL
LIN {X 0,Y 431.743,Z 781.39,A -85,B 0,C 180,E1 13469.785,E2 13469.785} C_VEL
LIN {X 0,Y 428.523,Z 810.016,A -85,B 0,C 180,E1 13469.295,E2 13469.295} C_VEL
LIN {X 0,Y 424.916,Z 832.209,A -85,B 0,C 180,E1 13468.805,E2 13468.805} C_VEL
LIN {X 0,Y 420.324,Z 854.729,A -85,B 0,C 180,E1 13468.167,E2 13468.167} C_VEL
LIN {X 0,Y 413.725,Z 880.591,A -85,B 0,C 180,E1 13467.248,E2 13467.248} C_VEL
LIN {X 0,Y 407.295,Z 901.672,A -85,B 0,C 180,E1 13466.325,E2 13466.325} C_VEL
LIN {X 0,Y 400.261,Z 921.948,A -85,B 0,C 180,E1 13465.27,E2 13465.27} C_VEL
LIN {X 0,Y 390.879,Z 945.835,A -85,B 0,C 180,E1 13463.778,E2 13463.778} C_VEL
LIN {X 0,Y 381.537,Z 966.672,A -85,B 0,C 180,E1 13462.196,E2 13462.196} C_VEL
LIN {X 0,Y 372.953,Z 984.235,A -85,B 0,C 180,E1 13460.629,E2 13460.629} C_VEL
LIN {X 0,Y 362.935,Z 1003.17,A -85,B 0,C 180,E1 13458.652,E2 13458.652} C_VEL
LIN {X 0,Y 351.732,Z 1022.499,A -85,B 0,C 180,E1 13456.223,E2 13456.223} C_VEL
LIN {X 0,Y 341.963,Z 1038.256,A -85,B 0,C 180,E1 13453.865,E2 13453.865} C_VEL
LIN {X 0,Y 332.737,Z 1052.415,A -85,B 0,C 180,E1 13451.383,E2 13451.383} C_VEL
LIN {X 0,Y 321.66,Z 1068.678,A -85,B 0,C 180,E1 13447.986,E2 13447.986} C_VEL
LIN {X 0,Y 312.045,Z 1082.135,A -85,B 0,C 180,E1 13444.551,E2 13444.551} C_VEL
LIN {X 0,Y 303.838,Z 1093.482,A -85,B 0,C 180,E1 13441.108,E2 13441.108} C_VEL
LIN {X 0,Y 295.289,Z 1105.397,A -85,B 0,C 180,E1 13436.766,E2 13436.766} C_VEL
LIN {X 0,Y 288.158,Z 1115.339,A -85,B 0,C 180,E1 13432.223,E2 13432.223} C_VEL
LIN {X 0,Y 283.131,Z 1122.782,A -85,B 0,C 180,E1 13428.105,E2 13428.105} C_VEL
LIN {X 0,Y 278.751,Z 1129.927,A -85,B 0,C 180,E1 13423.271,E2 13423.271} C_VEL
LIN {X 0,Y 275.536,Z 1135.935,A -85,B 0,C 180,E1 13417.926,E2 13417.926} C_VEL
LIN {X 0,Y 273.957,Z 1139.634,A -85,B 0,C 180,E1 13413.557,E2 13413.557} C_VEL
LIN {X 0,Y 273.134,Z 1142.239,A -85,B 0,C 180,E1 13409.371,E2 13409.371} C_VEL
LIN {X 0,Y 272.779,Z 1143.9,A -85,B 0,C 180,E1 13405.375,E2 13405.375} C_VEL
LIN {X 0,Y 272.712,Z 1144.778,A -85,B 0,C 180,E1 13401.354,E2 13401.354} C_VEL
LIN {X 0,Y 272.827,Z 1144.872,A -85,B 0,C 180,E1 13397.297,E2 13397.297} C_VEL
LIN {X 0,Y 273.201,Z 1144.165,A -85,B 0,C 180,E1 13393.194,E2 13393.194} C_VEL
LIN {X 0,Y 274.167,Z 1142.426,A -85,B 0,C 180,E1 13388.611,E2 13388.611} C_VEL
LIN {X 0,Y 276.703,Z 1138.609,A -85,B 0,C 180,E1 13382.683,E2 13382.683} C_VEL
LIN {X 0,Y 280.142,Z 1134.057,A -85,B 0,C 180,E1 13377.873,E2 13377.873} C_VEL
LIN {X 0,Y 284.761,Z 1128.523,A -85,B 0,C 180,E1 13373.351,E2 13373.351} C_VEL
LIN {X 0,Y 292.054,Z 1120.33,A -85,B 0,C 180,E1 13368.119,E2 13368.119} C_VEL
LIN {X 0,Y 300.401,Z 1111.039,A -85,B 0,C 180,E1 13363.552,E2 13363.552} C_VEL
LIN {X 0,Y 308.717,Z 1101.884,A -85,B 0,C 180,E1 13359.862,E2 13359.862} C_VEL
LIN {X 0,Y 320.121,Z 1089.239,A -85,B 0,C 180,E1 13355.7,E2 13355.7} C_VEL
LIN {X 0,Y 331.791,Z 1075.63,A -85,B 0,C 180,E1 13352.135,E2 13352.135} C_VEL
LIN {X 0,Y 342.168,Z 1063.098,A -85,B 0,C 180,E1 13349.402,E2 13349.402} C_VEL
LIN {X 0,Y 354.401,Z 1047.625,A -85,B 0,C 180,E1 13346.576,E2 13346.576} C_VEL
LIN {X 0,Y 367.482,Z 1029.659,A -85,B 0,C 180,E1 13343.907,E2 13343.907} C_VEL
LIN {X 0,Y 377.959,Z 1014.279,A -85,B 0,C 180,E1 13341.995,E2 13341.995} C_VEL
LIN {X 0,Y 388.437,Z 997.761,A -85,B 0,C 180,E1 13340.241,E2 13340.241} C_VEL
LIN {X 0,Y 401.215,Z 975.695,A -85,B 0,C 180,E1 13338.29,E2 13338.29} C_VEL
LIN {X 0,Y 401.876,Z 974.446,A -85,B 0,C 180,E1 13338.193,E2 13338.193} C_VEL
LIN {X 0,Y 404.743,Z 968.5,A -85,B 0,C 180,E1 13337.61,E2 13337.61} C_VEL
LIN {X 0,Y 408.679,Z 958.244,A -85,B 0,C 180,E1 13336.269,E2 13336.269} C_VEL
LIN {X 0,Y 411.254,Z 951.624,A -85,B 0,C 180,E1 13335.52,E2 13335.52} C_VEL
LIN {X 0,Y 412.933,Z 948.051,A -85,B 0,C 180,E1 13335.241,E2 13335.241} C_VEL
LIN {X 0,Y 422.982,Z 925.495,A -85,B 0,C 180,E1 13333.986,E2 13333.986} C_VEL
LIN {X 0,Y 430.619,Z 906.184,A -85,B 0,C 180,E1 13333.083,E2 13333.083} C_VEL
LIN {X 0,Y 437.712,Z 885.825,A -85,B 0,C 180,E1 13332.285,E2 13332.285} C_VEL
LIN {X 0,Y 444.878,Z 861.854,A -85,B 0,C 180,E1 13331.505,E2 13331.505} C_VEL
LIN {X 0,Y 450.738,Z 836.912,A -85,B 0,C 180,E1 13330.862,E2 13330.862} C_VEL
LIN {X 0,Y 454.844,Z 814.921,A -85,B 0,C 180,E1 13330.42,E2 13330.42} C_VEL
LIN {X 0,Y 458.201,Z 790.449,A -85,B 0,C 180,E1 13330.027,E2 13330.027} C_VEL
LIN {X 0,Y 480.365,Z 574.658,A -85,B 0,C 180,E1 13326.943,E2 13326.943} C_VEL
LIN {X 0,Y 478.371,Z 570.534,A -85,B 0,C 180,E1 13324.916,E2 13324.916} C_VEL
LIN {X 0,Y 476.678,Z 567.023,A -85,B 0,C 180,E1 13322.525,E2 13322.525} C_VEL
LIN {X 0,Y 475.368,Z 564.223,A -85,B 0,C 180,E1 13318.313,E2 13318.313} C_VEL
LIN {X 0,Y 475.467,Z 564.755,A -85,B 0,C 180,E1 13316.262,E2 13316.262} C_VEL
LIN {X 0,Y 476.999,Z 567.799,A -85,B 0,C 180,E1 13312.532,E2 13312.532} C_VEL
LIN {X 0,Y 479.062,Z 572.232,A -85,B 0,C 180,E1 13309.902,E2 13309.902} C_VEL
LIN {X 0,Y 480.93,Z 576.335,A -85,B 0,C 180,E1 13308.128,E2 13308.128} C_VEL
LIN {X 0,Y 458.285,Z 799.095,A -85,B 0,C 180,E1 13304.833,E2 13304.833} C_VEL
LIN {X 0,Y 454.816,Z 824.877,A -85,B 0,C 180,E1 13304.415,E2 13304.415} C_VEL
LIN {X 0,Y 450.66,Z 847.139,A -85,B 0,C 180,E1 13304.005,E2 13304.005} C_VEL
LIN {X 0,Y 444.73,Z 872.065,A -85,B 0,C 180,E1 13303.468,E2 13303.468} C_VEL
LIN {X 0,Y 436.919,Z 898.288,A -85,B 0,C 180,E1 13302.729,E2 13302.729} C_VEL
LIN {X 0,Y 429.46,Z 919.662,A -85,B 0,C 180,E1 13301.979,E2 13301.979} C_VEL
LIN {X 0,Y 421.585,Z 939.626,A -85,B 0,C 180,E1 13301.137,E2 13301.137} C_VEL
LIN {X 0,Y 411.362,Z 962.838,A -85,B 0,C 180,E1 13299.957,E2 13299.957} C_VEL
LIN {X 0,Y 399.414,Z 986.617,A -85,B 0,C 180,E1 13298.463,E2 13298.463} C_VEL
LIN {X 0,Y 389.266,Z 1005.038,A -85,B 0,C 180,E1 13297.081,E2 13297.081} C_VEL
LIN {X 0,Y 378.798,Z 1022.698,A -85,B 0,C 180,E1 13295.517,E2 13295.517} C_VEL
LIN {X 0,Y 366.488,Z 1042.075,A -85,B 0,C 180,E1 13293.49,E2 13293.49} C_VEL
LIN {X 0,Y 352.471,Z 1062.418,A -85,B 0,C 180,E1 13290.892,E2 13290.892} C_VEL
LIN {X 0,Y 341.195,Z 1077.911,A -85,B 0,C 180,E1 13288.514,E2 13288.514} C_VEL
LIN {X 0,Y 329.944,Z 1092.767,A -85,B 0,C 180,E1 13285.822,E2 13285.822} C_VEL
LIN {X 0,Y 317.248,Z 1109.091,A -85,B 0,C 180,E1 13282.285,E2 13282.285} C_VEL
LIN {X 0,Y 304.794,Z 1124.526,A -85,B 0,C 180,E1 13278.13,E2 13278.13} C_VEL
LIN {X 0,Y 295.662,Z 1135.95,A -85,B 0,C 180,E1 13274.429,E2 13274.429} C_VEL
LIN {X 0,Y 286.996,Z 1147.093,A -85,B 0,C 180,E1 13270.13,E2 13270.13} C_VEL
LIN {X 0,Y 278.08,Z 1159.184,A -85,B 0,C 180,E1 13264.368,E2 13264.368} C_VEL
LIN {X 0,Y 272.763,Z 1167.14,A -85,B 0,C 180,E1 13259.661,E2 13259.661} C_VEL
LIN {X 0,Y 269.042,Z 1173.571,A -85,B 0,C 180,E1 13255.066,E2 13255.066} C_VEL
LIN {X 0,Y 266.527,Z 1178.883,A -85,B 0,C 180,E1 13250.419,E2 13250.419} C_VEL
LIN {X 0,Y 265.1,Z 1183.097,A -85,B 0,C 180,E1 13245.757,E2 13245.757} C_VEL
LIN {X 0,Y 264.471,Z 1186.342,A -85,B 0,C 180,E1 13240.896,E2 13240.896} C_VEL
LIN {X 0,Y 264.434,Z 1188.463,A -85,B 0,C 180,E1 13235.86,E2 13235.86} C_VEL
LIN {X 0,Y 264.538,Z 1189.187,A -85,B 0,C 180,E1 13231.3,E2 13231.3} C_VEL
LIN {X 0,Y 264.523,Z 1188.705,A -85,B 0,C 180,E1 13226.75,E2 13226.75} C_VEL
LIN {X 0,Y 264.461,Z 1186.907,A -85,B 0,C 180,E1 13221.959,E2 13221.959} C_VEL
LIN {X 0,Y 264.692,Z 1183.828,A -85,B 0,C 180,E1 13217.123,E2 13217.123} C_VEL
LIN {X 0,Y 265.514,Z 1179.926,A -85,B 0,C 180,E1 13212.693,E2 13212.693} C_VEL
LIN {X 0,Y 267.225,Z 1174.767,A -85,B 0,C 180,E1 13208.119,E2 13208.119} C_VEL
LIN {X 0,Y 269.924,Z 1168.499,A -85,B 0,C 180,E1 13203.608,E2 13203.608} C_VEL
LIN {X 0,Y 274.134,Z 1160.416,A -85,B 0,C 180,E1 13198.807,E2 13198.807} C_VEL
LIN {X 0,Y 281.251,Z 1148.426,A -85,B 0,C 180,E1 13193.073,E2 13193.073} C_VEL
LIN {X 0,Y 287.921,Z 1137.989,A -85,B 0,C 180,E1 13188.979,E2 13188.979} C_VEL
LIN {X 0,Y 295.396,Z 1126.78,A -85,B 0,C 180,E1 13185.248,E2 13185.248} C_VEL
LIN {X 0,Y 305.246,Z 1112.305,A -85,B 0,C 180,E1 13181.179,E2 13181.179} C_VEL
LIN {X 0,Y 316.227,Z 1095.782,A -85,B 0,C 180,E1 13177.38,E2 13177.38} C_VEL
LIN {X 0,Y 326.152,Z 1080.566,A -85,B 0,C 180,E1 13174.447,E2 13174.447} C_VEL
LIN {X 0,Y 336.417,Z 1064.334,A -85,B 0,C 180,E1 13171.787,E2 13171.787} C_VEL
LIN {X 0,Y 349.506,Z 1042.412,A -85,B 0,C 180,E1 13168.807,E2 13168.807} C_VEL
LIN {X 0,Y 359.603,Z 1024.319,A -85,B 0,C 180,E1 13166.773,E2 13166.773} C_VEL
LIN {X 0,Y 369.116,Z 1006.161,A -85,B 0,C 180,E1 13165.03,E2 13165.03} C_VEL
LIN {X 0,Y 379.775,Z 984.244,A -85,B 0,C 180,E1 13163.244,E2 13163.244} C_VEL
LIN {X 0,Y 389.925,Z 960.754,A -85,B 0,C 180,E1 13161.67,E2 13161.67} C_VEL
LIN {X 0,Y 397.757,Z 940.755,A -85,B 0,C 180,E1 13160.55,E2 13160.55} C_VEL
LIN {X 0,Y 404.885,Z 920.523,A -85,B 0,C 180,E1 13159.592,E2 13159.592} C_VEL
LIN {X 0,Y 412.551,Z 895.906,A -85,B 0,C 180,E1 13158.626,E2 13158.626} C_VEL
LIN {X 0,Y 419.301,Z 869.489,A -85,B 0,C 180,E1 13157.816,E2 13157.816} C_VEL
LIN {X 0,Y 423.976,Z 847.4,A -85,B 0,C 180,E1 13157.285,E2 13157.285} C_VEL
LIN {X 0,Y 427.843,Z 823.803,A -85,B 0,C 180,E1 13156.808,E2 13156.808} C_VEL
LIN {X 0,Y 431.557,Z 787.998,A -85,B 0,C 180,E1 13156.206,E2 13156.206} C_VEL
LIN {X 0,Y 450.756,Z 566.742,A -85,B 0,C 180,E1 13152.781,E2 13152.781} C_VEL
LIN {X 0,Y 451.558,Z 556.786,A -85,B 0,C 180,E1 13152.598,E2 13152.598} C_VEL
LIN {X 0,Y 445.963,Z 545.682,A -85,B 0,C 180,E1 13149.811,E2 13149.811} C_VEL
LIN {X 0,Y 441.151,Z 536.621,A -85,B 0,C 180,E1 13146.965,E2 13146.965} C_VEL
LIN {X 0,Y 437.446,Z 529.838,A -85,B 0,C 180,E1 13144.26,E2 13144.26} C_VEL
LIN {X 0,Y 434.432,Z 524.411,A -85,B 0,C 180,E1 13141.451,E2 13141.451} C_VEL
LIN {X 0,Y 432.12,Z 520.191,A -85,B 0,C 180,E1 13138.334,E2 13138.334} C_VEL
LIN {X 0,Y 430.527,Z 517.666,A -85,B 0,C 180,E1 13133.713,E2 13133.713} C_VEL
LIN {X 0,Y 430.69,Z 518.097,A -85,B 0,C 180,E1 13130.782,E2 13130.782} C_VEL
LIN {X 0,Y 432.47,Z 520.734,A -85,B 0,C 180,E1 13126.739,E2 13126.739} C_VEL
LIN {X 0,Y 435.034,Z 525.411,A -85,B 0,C 180,E1 13123.578,E2 13123.578} C_VEL
LIN {X 0,Y 438.624,Z 531.687,A -85,B 0,C 180,E1 13120.49,E2 13120.49} C_VEL
LIN {X 0,Y 443.169,Z 540.231,A -85,B 0,C 180,E1 13117.446,E2 13117.446} C_VEL
LIN {X 0,Y 447.852,Z 549.356,A -85,B 0,C 180,E1 13114.864,E2 13114.864} C_VEL
LIN {X 0,Y 449.092,Z 552.022,A -85,B 0,C 180,E1 13114.236,E2 13114.236} C_VEL
LIN {X 0,Y 428.104,Z 788.034,A -85,B 0,C 180,E1 13110.67,E2 13110.67} C_VEL
LIN {X 0,Y 425.126,Z 812.367,A -85,B 0,C 180,E1 13110.243,E2 13110.243} C_VEL
LIN {X 0,Y 421.358,Z 834.674,A -85,B 0,C 180,E1 13109.748,E2 13109.748} C_VEL
LIN {X 0,Y 415.635,Z 861.168,A -85,B 0,C 180,E1 13108.981,E2 13108.981} C_VEL
LIN {X 0,Y 409.595,Z 883.524,A -85,B 0,C 180,E1 13108.157,E2 13108.157} C_VEL
LIN {X 0,Y 403.469,Z 903.088,A -85,B 0,C 180,E1 13107.299,E2 13107.299} C_VEL
LIN {X 0,Y 396.254,Z 923.394,A -85,B 0,C 180,E1 13106.245,E2 13106.245} C_VEL
LIN {X 0,Y 386.063,Z 948.468,A -85,B 0,C 180,E1 13104.668,E2 13104.668} C_VEL
LIN {X 0,Y 377.132,Z 967.9,A -85,B 0,C 180,E1 13103.188,E2 13103.188} C_VEL
LIN {X 0,Y 368.143,Z 985.823,A -85,B 0,C 180,E1 13101.587,E2 13101.587} C_VEL
LIN {X 0,Y 356.859,Z 1006.489,A -85,B 0,C 180,E1 13099.402,E2 13099.402} C_VEL
LIN {X 0,Y 346.341,Z 1023.994,A -85,B 0,C 180,E1 13097.162,E2 13097.162} C_VEL
LIN {X 0,Y 336.903,Z 1038.795,A -85,B 0,C 180,E1 13094.937,E2 13094.937} C_VEL
LIN {X 0,Y 327.398,Z 1052.96,A -85,B 0,C 180,E1 13092.448,E2 13092.448} C_VEL
LIN {X 0,Y 315.96,Z 1069.24,A -85,B 0,C 180,E1 13089.03,E2 13089.03} C_VEL
LIN {X 0,Y 305.84,Z 1082.919,A -85,B 0,C 180,E1 13085.505,E2 13085.505} C_VEL
LIN {X 0,Y 297.468,Z 1094.062,A -85,B 0,C 180,E1 13082.078,E2 13082.078} C_VEL
LIN {X 0,Y 288.555,Z 1105.988,A -85,B 0,C 180,E1 13077.666,E2 13077.666} C_VEL
LIN {X 0,Y 281.083,Z 1115.943,A -85,B 0,C 180,E1 13073.034,E2 13073.034} C_VEL
LIN {X 0,Y 275.8,Z 1123.391,A -85,B 0,C 180,E1 13068.823,E2 13068.823} C_VEL
LIN {X 0,Y 271.17,Z 1130.541,A -85,B 0,C 180,E1 13063.867,E2 13063.867} C_VEL
LIN {X 0,Y 267.757,Z 1136.558,A -85,B 0,C 180,E1 13058.374,E2 13058.374} C_VEL
LIN {X 0,Y 266.011,Z 1140.413,A -85,B 0,C 180,E1 13053.663,E2 13053.663} C_VEL
LIN {X 0,Y 265.16,Z 1142.983,A -85,B 0,C 180,E1 13049.352,E2 13049.352} C_VEL
LIN {X 0,Y 264.793,Z 1144.678,A -85,B 0,C 180,E1 13045.018,E2 13045.018} C_VEL
LIN {X 0,Y 264.736,Z 1145.486,A -85,B 0,C 180,E1 13040.873,E2 13040.873} C_VEL
LIN {X 0,Y 264.901,Z 1145.497,A -85,B 0,C 180,E1 13036.466,E2 13036.466} C_VEL
LIN {X 0,Y 265.591,Z 1144.404,A -85,B 0,C 180,E1 13031.109,E2 13031.109} C_VEL
LIN {X 0,Y 267.313,Z 1141.644,A -85,B 0,C 180,E1 13025.469,E2 13025.469} C_VEL
LIN {X 0,Y 269.919,Z 1138.192,A -85,B 0,C 180,E1 13020.727,E2 13020.727} C_VEL
LIN {X 0,Y 274.006,Z 1133.373,A -85,B 0,C 180,E1 13015.809,E2 13015.809} C_VEL
LIN {X 0,Y 280.776,Z 1125.905,A -85,B 0,C 180,E1 13010.134,E2 13010.134} C_VEL
LIN {X 0,Y 287.932,Z 1118.298,A -85,B 0,C 180,E1 13005.674,E2 13005.674} C_VEL
LIN {X 0,Y 296.355,Z 1109.508,A -85,B 0,C 180,E1 13001.496,E2 13001.496} C_VEL
LIN {X 0,Y 308.25,Z 1096.911,A -85,B 0,C 180,E1 12996.757,E2 12996.757} C_VEL
LIN {X 0,Y 318.509,Z 1085.727,A -85,B 0,C 180,E1 12993.382,E2 12993.382} C_VEL
LIN {X 0,Y 329.131,Z 1073.757,A -85,B 0,C 180,E1 12990.373,E2 12990.373} C_VEL
LIN {X 0,Y 342.552,Z 1057.856,A -85,B 0,C 180,E1 12987.088,E2 12987.088} C_VEL
LIN {X 0,Y 354.821,Z 1042.213,A -85,B 0,C 180,E1 12984.468,E2 12984.468} C_VEL
LIN {X 0,Y 366.19,Z 1026.803,A -85,B 0,C 180,E1 12982.305,E2 12982.305} C_VEL
LIN {X 0,Y 379.536,Z 1007.332,A -85,B 0,C 180,E1 12980.029,E2 12980.029} C_VEL
LIN {X 0,Y 391.679,Z 987.62,A -85,B 0,C 180,E1 12978.146,E2 12978.146} C_VEL
LIN {X 0,Y 401.487,Z 970.299,A -85,B 0,C 180,E1 12976.753,E2 12976.753} C_VEL
LIN {X 0,Y 411.299,Z 951.282,A -85,B 0,C 180,E1 12975.446,E2 12975.446} C_VEL
LIN {X 0,Y 412.933,Z 948.051,A -85,B 0,C 180,E1 12975.241,E2 12975.241} C_VEL
LIN {X 0,Y 415.681,Z 941.809,A -85,B 0,C 180,E1 12974.728,E2 12974.728} C_VEL
LIN {X 0,Y 420.741,Z 926.425,A -85,B 0,C 180,E1 12973.094,E2 12973.094} C_VEL
LIN {X 0,Y 423.23,Z 919.885,A -85,B 0,C 180,E1 12972.643,E2 12972.643} C_VEL
LIN {X 0,Y 432.751,Z 894.934,A -85,B 0,C 180,E1 12971.582,E2 12971.582} C_VEL
LIN {X 0,Y 439.757,Z 873.047,A -85,B 0,C 180,E1 12970.82,E2 12970.82} C_VEL
LIN {X 0,Y 445.673,Z 851.23,A -85,B 0,C 180,E1 12970.201,E2 12970.201} C_VEL
LIN {X 0,Y 450.878,Z 827.83,A -85,B 0,C 180,E1 12969.673,E2 12969.673} C_VEL
LIN {X 0,Y 455.262,Z 800.571,A -85,B 0,C 180,E1 12969.196,E2 12969.196} C_VEL
LIN {X 0,Y 466.211,Z 696.828,A -85,B 0,C 180,E1 12967.709,E2 12967.709} C_VEL
LIN {X 0,Y 478.421,Z 580.874,A -85,B 0,C 180,E1 12966.059,E2 12966.059} C_VEL
LIN {X 0,Y 476.968,Z 577.888,A -85,B 0,C 180,E1 12964.449,E2 12964.449} C_VEL
LIN {X 0,Y 475.624,Z 574.902,A -85,B 0,C 180,E1 12962.41,E2 12962.41} C_VEL
LIN {X 0,Y 474.385,Z 572.138,A -85,B 0,C 180,E1 12958.188,E2 12958.188} C_VEL
LIN {X 0,Y 474.526,Z 572.884,A -85,B 0,C 180,E1 12956.013,E2 12956.013} C_VEL
LIN {X 0,Y 475.934,Z 575.705,A -85,B 0,C 180,E1 12952.637,E2 12952.637} C_VEL
LIN {X 0,Y 477.898,Z 580.055,A -85,B 0,C 180,E1 12950.06,E2 12950.06} C_VEL
LIN {X 0,Y 478.939,Z 582.479,A -85,B 0,C 180,E1 12948.984,E2 12948.984} C_VEL
LIN {X 0,Y 456.016,Z 802.986,A -85,B 0,C 180,E1 12945.754,E2 12945.754} C_VEL
LIN {X 0,Y 452.753,Z 826.073,A -85,B 0,C 180,E1 12945.38,E2 12945.38} C_VEL
LIN {X 0,Y 448.322,Z 849.032,A -85,B 0,C 180,E1 12944.963,E2 12944.963} C_VEL
LIN {X 0,Y 441.296,Z 876.976,A -85,B 0,C 180,E1 12944.352,E2 12944.352} C_VEL
LIN {X 0,Y 434.365,Z 899.367,A -85,B 0,C 180,E1 12943.716,E2 12943.716} C_VEL
LIN {X 0,Y 427.081,Z 919.796,A -85,B 0,C 180,E1 12943.01,E2 12943.01} C_VEL
LIN {X 0,Y 418.622,Z 940.784,A -85,B 0,C 180,E1 12942.138,E2 12942.138} C_VEL
LIN {X 0,Y 406.84,Z 966.527,A -85,B 0,C 180,E1 12940.821,E2 12940.821} C_VEL
LIN {X 0,Y 396.417,Z 986.704,A -85,B 0,C 180,E1 12939.556,E2 12939.556} C_VEL
LIN {X 0,Y 386.07,Z 1005.062,A -85,B 0,C 180,E1 12938.195,E2 12938.195} C_VEL
LIN {X 0,Y 374.85,Z 1023.528,A -85,B 0,C 180,E1 12936.574,E2 12936.574} C_VEL
LIN {X 0,Y 360.647,Z 1045.088,A -85,B 0,C 180,E1 12934.294,E2 12934.294} C_VEL
LIN {X 0,Y 347.779,Z 1063.098,A -85,B 0,C 180,E1 12931.96,E2 12931.96} C_VEL
LIN {X 0,Y 336.566,Z 1078.022,A -85,B 0,C 180,E1 12929.665,E2 12929.665} C_VEL
LIN {X 0,Y 325.144,Z 1092.593,A -85,B 0,C 180,E1 12927.022,E2 12927.022} C_VEL
LIN {X 0,Y 311.57,Z 1109.386,A -85,B 0,C 180,E1 12923.348,E2 12923.348} C_VEL
LIN {X 0,Y 299.157,Z 1124.145,A -85,B 0,C 180,E1 12919.325,E2 12919.325} C_VEL
LIN {X 0,Y 289.652,Z 1135.493,A -85,B 0,C 180,E1 12915.606,E2 12915.606} C_VEL
LIN {X 0,Y 280.495,Z 1146.672,A -85,B 0,C 180,E1 12911.222,E2 12911.222} C_VEL
LIN {X 0,Y 271.128,Z 1158.651,A -85,B 0,C 180,E1 12905.379,E2 12905.379} C_VEL
LIN {X 0,Y 265.479,Z 1166.585,A -85,B 0,C 180,E1 12900.56,E2 12900.56} C_VEL
LIN {X 0,Y 261.483,Z 1172.996,A -85,B 0,C 180,E1 12895.844,E2 12895.844} C_VEL
LIN {X 0,Y 258.775,Z 1178.292,A -85,B 0,C 180,E1 12891.059,E2 12891.059} C_VEL
LIN {X 0,Y 257.154,Z 1182.671,A -85,B 0,C 180,E1 12886.025,E2 12886.025} C_VEL
LIN {X 0,Y 256.459,Z 1186.245,A -85,B 0,C 180,E1 12880.331,E2 12880.331} C_VEL
LIN {X 0,Y 256.478,Z 1188.016,A -85,B 0,C 180,E1 12875.144,E2 12875.144} C_VEL
LIN {X 0,Y 256.571,Z 1188.477,A -85,B 0,C 180,E1 12870.67,E2 12870.67} C_VEL
LIN {X 0,Y 256.54,Z 1187.867,A -85,B 0,C 180,E1 12866.19,E2 12866.19} C_VEL
LIN {X 0,Y 256.484,Z 1186.062,A -85,B 0,C 180,E1 12861.481,E2 12861.481} C_VEL
LIN {X 0,Y 256.748,Z 1183.076,A -85,B 0,C 180,E1 12856.717,E2 12856.717} C_VEL
LIN {X 0,Y 257.649,Z 1179.142,A -85,B 0,C 180,E1 12852.147,E2 12852.147} C_VEL
LIN {X 0,Y 259.446,Z 1174.12,A -85,B 0,C 180,E1 12847.572,E2 12847.572} C_VEL
LIN {X 0,Y 262.262,Z 1167.977,A -85,B 0,C 180,E1 12843.02,E2 12843.02} C_VEL
LIN {X 0,Y 266.46,Z 1160.299,A -85,B 0,C 180,E1 12838.31,E2 12838.31} C_VEL
LIN {X 0,Y 273.534,Z 1148.957,A -85,B 0,C 180,E1 12832.643,E2 12832.643} C_VEL
LIN {X 0,Y 280.758,Z 1138.092,A -85,B 0,C 180,E1 12828.244,E2 12828.244} C_VEL
LIN {X 0,Y 288.513,Z 1126.934,A -85,B 0,C 180,E1 12824.432,E2 12824.432} C_VEL
LIN {X 0,Y 297.28,Z 1114.475,A -85,B 0,C 180,E1 12820.821,E2 12820.821} C_VEL
LIN {X 0,Y 308.985,Z 1097.706,A -85,B 0,C 180,E1 12816.775,E2 12816.775} C_VEL
LIN {X 0,Y 320.162,Z 1081.112,A -85,B 0,C 180,E1 12813.506,E2 12813.506} C_VEL
LIN {X 0,Y 330.054,Z 1065.969,A -85,B 0,C 180,E1 12810.984,E2 12810.984} C_VEL
LIN {X 0,Y 341.193,Z 1048.146,A -85,B 0,C 180,E1 12808.461,E2 12808.461} C_VEL
LIN {X 0,Y 353.985,Z 1026.117,A -85,B 0,C 180,E1 12805.891,E2 12805.891} C_VEL
LIN {X 0,Y 363.748,Z 1008.039,A -85,B 0,C 180,E1 12804.135,E2 12804.135} C_VEL
LIN {X 0,Y 372.688,Z 990.227,A -85,B 0,C 180,E1 12802.648,E2 12802.648} C_VEL
LIN {X 0,Y 382.646,Z 968.695,A -85,B 0,C 180,E1 12801.118,E2 12801.118} C_VEL
LIN {X 0,Y 393.12,Z 943.158,A -85,B 0,C 180,E1 12799.638,E2 12799.638} C_VEL
LIN {X 0,Y 400.515,Z 922.827,A -85,B 0,C 180,E1 12798.667,E2 12798.667} C_VEL
LIN {X 0,Y 407.236,Z 902.001,A -85,B 0,C 180,E1 12797.834,E2 12797.834} C_VEL
LIN {X 0,Y 414.336,Z 876.652,A -85,B 0,C 180,E1 12797.006,E2 12797.006} C_VEL
LIN {X 0,Y 420.268,Z 849.964,A -85,B 0,C 180,E1 12796.343,E2 12796.343} C_VEL
LIN {X 0,Y 424.143,Z 827.57,A -85,B 0,C 180,E1 12795.888,E2 12795.888} C_VEL
LIN {X 0,Y 427.116,Z 803.298,A -85,B 0,C 180,E1 12795.459,E2 12795.459} C_VEL
LIN {X 0,Y 446.921,Z 580.332,A -85,B 0,C 180,E1 12792.021,E2 12792.021} C_VEL
LIN {X 0,Y 448.581,Z 561.91,A -85,B 0,C 180,E1 12791.736,E2 12791.736} C_VEL
LIN {X 0,Y 443.594,Z 551.778,A -85,B 0,C 180,E1 12789.111,E2 12789.111} C_VEL
LIN {X 0,Y 439.255,Z 543.416,A -85,B 0,C 180,E1 12786.404,E2 12786.404} C_VEL
LIN {X 0,Y 435.656,Z 536.588,A -85,B 0,C 180,E1 12783.619,E2 12783.619} C_VEL
LIN {X 0,Y 433.064,Z 531.935,A -85,B 0,C 180,E1 12781.058,E2 12781.058} C_VEL
LIN {X 0,Y 431.095,Z 528.112,A -85,B 0,C 180,E1 12778.272,E2 12778.272} C_VEL
LIN {X 0,Y 429.539,Z 525.586,A -85,B 0,C 180,E1 12773.585,E2 12773.585} C_VEL
LIN {X 0,Y 429.715,Z 526.057,A -85,B 0,C 180,E1 12770.761,E2 12770.761} C_VEL
LIN {X 0,Y 431.355,Z 528.513,A -85,B 0,C 180,E1 12766.938,E2 12766.938} C_VEL
LIN {X 0,Y 433.866,Z 533.26,A -85,B 0,C 180,E1 12763.739,E2 12763.739} C_VEL
LIN {X 0,Y 437.219,Z 539.269,A -85,B 0,C 180,E1 12760.772,E2 12760.772} C_VEL
LIN {X 0,Y 441.601,Z 547.74,A -85,B 0,C 180,E1 12757.747,E2 12757.747} C_VEL
LIN {X 0,Y 446.09,Z 556.754,A -85,B 0,C 180,E1 12755.197,E2 12755.197} C_VEL
LIN {X 0,Y 446.152,Z 557.469,A -85,B 0,C 180,E1 12755.134,E2 12755.134} C_VEL
LIN {X 0,Y 424.829,Z 791.563,A -85,B 0,C 180,E1 12751.618,E2 12751.618} C_VEL
LIN {X 0,Y 421.943,Z 814.086,A -85,B 0,C 180,E1 12751.22,E2 12751.22} C_VEL
LIN {X 0,Y 417.825,Z 837.635,A -85,B 0,C 180,E1 12750.695,E2 12750.695} C_VEL
LIN {X 0,Y 411.704,Z 864.465,A -85,B 0,C 180,E1 12749.903,E2 12749.903} C_VEL
LIN {X 0,Y 405.943,Z 885.209,A -85,B 0,C 180,E1 12749.134,E2 12749.134} C_VEL
LIN {X 0,Y 399.66,Z 904.771,A -85,B 0,C 180,E1 12748.277,E2 12748.277} C_VEL
LIN {X 0,Y 391.195,Z 927.948,A -85,B 0,C 180,E1 12747.065,E2 12747.065} C_VEL
LIN {X 0,Y 381.615,Z 950.506,A -85,B 0,C 180,E1 12745.621,E2 12745.621} C_VEL
LIN {X 0,Y 372.911,Z 968.993,A -85,B 0,C 180,E1 12744.214,E2 12744.214} C_VEL
LIN {X 0,Y 363.677,Z 986.961,A -85,B 0,C 180,E1 12742.612,E2 12742.612} C_VEL
LIN {X 0,Y 351.804,Z 1008.056,A -85,B 0,C 180,E1 12740.372,E2 12740.372} C_VEL
LIN {X 0,Y 341.045,Z 1025.482,A -85,B 0,C 180,E1 12738.13,E2 12738.13} C_VEL
LIN {X 0,Y 331.375,Z 1040.213,A -85,B 0,C 180,E1 12735.899,E2 12735.899} C_VEL
LIN {X 0,Y 319.964,Z 1056.71,A -85,B 0,C 180,E1 12732.94,E2 12732.94} C_VEL
LIN {X 0,Y 308.313,Z 1072.446,A -85,B 0,C 180,E1 12729.466,E2 12729.466} C_VEL
LIN {X 0,Y 299.119,Z 1084.474,A -85,B 0,C 180,E1 12726.274,E2 12726.274} C_VEL
LIN {X 0,Y 289.949,Z 1096.261,A -85,B 0,C 180,E1 12722.544,E2 12722.544} C_VEL
LIN {X 0,Y 280.12,Z 1108.727,A -85,B 0,C 180,E1 12717.647,E2 12717.647} C_VEL
LIN {X 0,Y 273.487,Z 1117.296,A -85,B 0,C 180,E1 12713.484,E2 12713.484} C_VEL
LIN {X 0,Y 267.816,Z 1124.985,A -85,B 0,C 180,E1 12708.953,E2 12708.953} C_VEL
LIN {X 0,Y 262.476,Z 1132.917,A -85,B 0,C 180,E1 12702.988,E2 12702.988} C_VEL
LIN {X 0,Y 259.673,Z 1137.758,A -85,B 0,C 180,E1 12698.19,E2 12698.19} C_VEL
LIN {X 0,Y 257.998,Z 1141.342,A -85,B 0,C 180,E1 12693.555,E2 12693.555} C_VEL
LIN {X 0,Y 257.131,Z 1143.942,A -85,B 0,C 180,E1 12688.886,E2 12688.886} C_VEL
LIN {X 0,Y 256.781,Z 1145.799,A -85,B 0,C 180,E1 12683.516,E2 12683.516} C_VEL
LIN {X 0,Y 256.827,Z 1146.293,A -85,B 0,C 180,E1 12678.32,E2 12678.32} C_VEL
LIN {X 0,Y 257.222,Z 1145.749,A -85,B 0,C 180,E1 12673.515,E2 12673.515} C_VEL
LIN {X 0,Y 258.145,Z 1144.312,A -85,B 0,C 180,E1 12668.887,E2 12668.887} C_VEL
LIN {X 0,Y 259.917,Z 1141.893,A -85,B 0,C 180,E1 12664.183,E2 12664.183} C_VEL
LIN {X 0,Y 262.964,Z 1138.256,A -85,B 0,C 180,E1 12659.243,E2 12659.243} C_VEL
LIN {X 0,Y 268.962,Z 1131.756,A -85,B 0,C 180,E1 12652.97,E2 12652.97} C_VEL
LIN {X 0,Y 275.211,Z 1125.329,A -85,B 0,C 180,E1 12648.329,E2 12648.329} C_VEL
LIN {X 0,Y 282.529,Z 1118.006,A -85,B 0,C 180,E1 12644.077,E2 12644.077} C_VEL
LIN {X 0,Y 293.061,Z 1107.567,A -85,B 0,C 180,E1 12639.243,E2 12639.243} C_VEL
LIN {X 0,Y 304.244,Z 1096.077,A -85,B 0,C 180,E1 12635.084,E2 12635.084} C_VEL
LIN {X 0,Y 315.046,Z 1084.726,A -85,B 0,C 180,E1 12631.728,E2 12631.728} C_VEL
LIN {X 0,Y 328.747,Z 1069.671,A -85,B 0,C 180,E1 12628.114,E2 12628.114} C_VEL
LIN {X 0,Y 340.799,Z 1055.47,A -85,B 0,C 180,E1 12625.36,E2 12625.36} C_VEL
LIN {X 0,Y 352.11,Z 1041.368,A -85,B 0,C 180,E1 12623.068,E2 12623.068} C_VEL
LIN {X 0,Y 364.696,Z 1024.638,A -85,B 0,C 180,E1 12620.789,E2 12620.789} C_VEL
LIN {X 0,Y 378.583,Z 1004.368,A -85,B 0,C 180,E1 12618.533,E2 12618.533} C_VEL
LIN {X 0,Y 389.346,Z 987.161,A -85,B 0,C 180,E1 12616.943,E2 12616.943} C_VEL
LIN {X 0,Y 399.94,Z 968.697,A -85,B 0,C 180,E1 12615.499,E2 12615.499} C_VEL
LIN {X 0,Y 411.69,Z 945.855,A -85,B 0,C 180,E1 12614.01,E2 12614.01} C_VEL
LIN {X 0,Y 420.962,Z 925.261,A -85,B 0,C 180,E1 12612.901,E2 12612.901} C_VEL
LIN {X 0,Y 423.23,Z 919.885,A -85,B 0,C 180,E1 12612.643,E2 12612.643} C_VEL
LIN {X 0,Y 425.719,Z 913.277,A -85,B 0,C 180,E1 12612.207,E2 12612.207} C_VEL
LIN {X 0,Y 430.456,Z 897.057,A -85,B 0,C 180,E1 12610.747,E2 12610.747} C_VEL
LIN {X 0,Y 432.537,Z 890.198,A -85,B 0,C 180,E1 12610.36,E2 12610.36} C_VEL
LIN {X 0,Y 438.569,Z 871.259,A -85,B 0,C 180,E1 12609.735,E2 12609.735} C_VEL
LIN {X 0,Y 444.652,Z 848.759,A -85,B 0,C 180,E1 12609.12,E2 12609.12} C_VEL
LIN {X 0,Y 450.601,Z 820.522,A -85,B 0,C 180,E1 12608.53,E2 12608.53} C_VEL
LIN {X 0,Y 454.036,Z 797.924,A -85,B 0,C 180,E1 12608.163,E2 12608.163} C_VEL
LIN {X 0,Y 476.621,Z 587.263,A -85,B 0,C 180,E1 12605.213,E2 12605.213} C_VEL
LIN {X 0,Y 474.573,Z 582.781,A -85,B 0,C 180,E1 12602.294,E2 12602.294} C_VEL
LIN {X 0,Y 473.403,Z 580.079,A -85,B 0,C 180,E1 12598.184,E2 12598.184} C_VEL
LIN {X 0,Y 473.522,Z 580.771,A -85,B 0,C 180,E1 12596.125,E2 12596.125} C_VEL
LIN {X 0,Y 474.836,Z 583.511,A -85,B 0,C 180,E1 12592.802,E2 12592.802} C_VEL
LIN {X 0,Y 476.685,Z 587.75,A -85,B 0,C 180,E1 12590.279,E2 12590.279} C_VEL
LIN {X 0,Y 477.051,Z 588.858,A -85,B 0,C 180,E1 12589.845,E2 12589.845} C_VEL
LIN {X 0,Y 454.111,Z 804.926,A -85,B 0,C 180,E1 12586.714,E2 12586.714} C_VEL
LIN {X 0,Y 450.818,Z 827.277,A -85,B 0,C 180,E1 12586.355,E2 12586.355} C_VEL
LIN {X 0,Y 445.499,Z 853.785,A -85,B 0,C 180,E1 12585.876,E2 12585.876} C_VEL
LIN {X 0,Y 438.545,Z 879.688,A -85,B 0,C 180,E1 12585.3,E2 12585.3} C_VEL
LIN {X 0,Y 431.92,Z 900.528,A -85,B 0,C 180,E1 12584.712,E2 12584.712} C_VEL
LIN {X 0,Y 424.368,Z 921.203,A -85,B 0,C 180,E1 12584.007,E2 12584.007} C_VEL
LIN {X 0,Y 414.095,Z 945.935,A -85,B 0,C 180,E1 12582.973,E2 12582.973} C_VEL
LIN {X 0,Y 402.721,Z 969.505,A -85,B 0,C 180,E1 12581.742,E2 12581.742} C_VEL
LIN {X 0,Y 392.901,Z 987.999,A -85,B 0,C 180,E1 12580.582,E2 12580.582} C_VEL
LIN {X 0,Y 381.894,Z 1007.003,A -85,B 0,C 180,E1 12579.177,E2 12579.177} C_VEL
LIN {X 0,Y 367.757,Z 1029.367,A -85,B 0,C 180,E1 12577.172,E2 12577.172} C_VEL
LIN {X 0,Y 354.402,Z 1048.604,A -85,B 0,C 180,E1 12575.05,E2 12575.05} C_VEL
LIN {X 0,Y 342.498,Z 1064.731,A -85,B 0,C 180,E1 12572.922,E2 12572.922} C_VEL
LIN {X 0,Y 329.339,Z 1081.64,A -85,B 0,C 180,E1 12570.26,E2 12570.26} C_VEL
LIN {X 0,Y 314.435,Z 1099.69,A -85,B 0,C 180,E1 12566.752,E2 12566.752} C_VEL
LIN {X 0,Y 302.873,Z 1113.182,A -85,B 0,C 180,E1 12563.541,E2 12563.541} C_VEL
LIN {X 0,Y 292.166,Z 1125.466,A -85,B 0,C 180,E1 12560.048,E2 12560.048} C_VEL
LIN {X 0,Y 280.392,Z 1139.045,A -85,B 0,C 180,E1 12555.371,E2 12555.371} C_VEL
LIN {X 0,Y 269.997,Z 1151.076,A -85,B 0,C 180,E1 12550.118,E2 12550.118} C_VEL
LIN {X 0,Y 263.061,Z 1159.638,A -85,B 0,C 180,E1 12545.558,E2 12545.558} C_VEL
LIN {X 0,Y 257.332,Z 1167.35,A -85,B 0,C 180,E1 12540.597,E2 12540.597} C_VEL
LIN {X 0,Y 252.421,Z 1175.158,A -85,B 0,C 180,E1 12534.328,E2 12534.328} C_VEL
LIN {X 0,Y 249.75,Z 1180.634,A -85,B 0,C 180,E1 12528.404,E2 12528.404} C_VEL
LIN {X 0,Y 248.742,Z 1183.909,A -85,B 0,C 180,E1 12523.719,E2 12523.719} C_VEL
LIN {X 0,Y 248.447,Z 1186.212,A -85,B 0,C 180,E1 12519.03,E2 12519.03} C_VEL
LIN {X 0,Y 248.518,Z 1187.464,A -85,B 0,C 180,E1 12514.615,E2 12514.615} C_VEL
LIN {X 0,Y 248.603,Z 1187.789,A -85,B 0,C 180,E1 12510.461,E2 12510.461} C_VEL
LIN {X 0,Y 248.564,Z 1187.17,A -85,B 0,C 180,E1 12506.053,E2 12506.053} C_VEL
LIN {X 0,Y 248.504,Z 1185.467,A -85,B 0,C 180,E1 12501.439,E2 12501.439} C_VEL
LIN {X 0,Y 248.783,Z 1182.502,A -85,B 0,C 180,E1 12496.52,E2 12496.52} C_VEL
LIN {X 0,Y 249.74,Z 1178.585,A -85,B 0,C 180,E1 12491.803,E2 12491.803} C_VEL
LIN {X 0,Y 251.641,Z 1173.577,A -85,B 0,C 180,E1 12487.084,E2 12487.084} C_VEL
LIN {X 0,Y 254.624,Z 1167.454,A -85,B 0,C 180,E1 12482.396,E2 12482.396} C_VEL
LIN {X 0,Y 259.045,Z 1159.793,A -85,B 0,C 180,E1 12477.554,E2 12477.554} C_VEL
LIN {X 0,Y 266.151,Z 1148.981,A -85,B 0,C 180,E1 12471.968,E2 12471.968} C_VEL
LIN {X 0,Y 274.44,Z 1137.079,A -85,B 0,C 180,E1 12467.056,E2 12467.056} C_VEL
LIN {X 0,Y 282.553,Z 1125.905,A -85,B 0,C 180,E1 12463.201,E2 12463.201} C_VEL
LIN {X 0,Y 292.667,Z 1112.11,A -85,B 0,C 180,E1 12459.202,E2 12459.202} C_VEL
LIN {X 0,Y 304.742,Z 1095.278,A -85,B 0,C 180,E1 12455.218,E2 12455.218} C_VEL
LIN {X 0,Y 315.185,Z 1080.289,A -85,B 0,C 180,E1 12452.284,E2 12452.284} C_VEL
LIN {X 0,Y 325.383,Z 1065.123,A -85,B 0,C 180,E1 12449.764,E2 12449.764} C_VEL
LIN {X 0,Y 337.497,Z 1046.252,A -85,B 0,C 180,E1 12447.114,E2 12447.114} C_VEL
LIN {X 0,Y 349.968,Z 1025.185,A -85,B 0,C 180,E1 12444.698,E2 12444.698} C_VEL
LIN {X 0,Y 359.88,Z 1007.227,A -85,B 0,C 180,E1 12442.973,E2 12442.973} C_VEL
LIN {X 0,Y 369.113,Z 989.221,A -85,B 0,C 180,E1 12441.491,E2 12441.491} C_VEL
LIN {X 0,Y 379.677,Z 966.79,A -85,B 0,C 180,E1 12439.926,E2 12439.926} C_VEL
LIN {X 0,Y 389.764,Z 942.473,A -85,B 0,C 180,E1 12438.549,E2 12438.549} C_VEL
LIN {X 0,Y 397.485,Z 921.545,A -85,B 0,C 180,E1 12437.568,E2 12437.568} C_VEL
LIN {X 0,Y 404.381,Z 900.429,A -85,B 0,C 180,E1 12436.744,E2 12436.744} C_VEL
LIN {X 0,Y 411.913,Z 873.433,A -85,B 0,C 180,E1 12435.896,E2 12435.896} C_VEL
LIN {X 0,Y 417.431,Z 848.67,A -85,B 0,C 180,E1 12435.304,E2 12435.304} C_VEL
LIN {X 0,Y 421.303,Z 826.412,A -85,B 0,C 180,E1 12434.858,E2 12434.858} C_VEL
LIN {X 0,Y 424.553,Z 799.81,A -85,B 0,C 180,E1 12434.396,E2 12434.396} C_VEL
LIN {X 0,Y 444.819,Z 575.964,A -85,B 0,C 180,E1 12430.974,E2 12430.974} C_VEL
LIN {X 0,Y 445.645,Z 566.898,A -85,B 0,C 180,E1 12430.831,E2 12430.831} C_VEL
LIN {X 0,Y 440.97,Z 557.299,A -85,B 0,C 180,E1 12428.213,E2 12428.213} C_VEL
LIN {X 0,Y 437.038,Z 549.624,A -85,B 0,C 180,E1 12425.58,E2 12425.58} C_VEL
LIN {X 0,Y 434.055,Z 543.665,A -85,B 0,C 180,E1 12423.103,E2 12423.103} C_VEL
LIN {X 0,Y 431.831,Z 539.627,A -85,B 0,C 180,E1 12420.796,E2 12420.796} C_VEL
LIN {X 0,Y 430.026,Z 535.985,A -85,B 0,C 180,E1 12418.135,E2 12418.135} C_VEL
LIN {X 0,Y 428.56,Z 533.525,A -85,B 0,C 180,E1 12413.57,E2 12413.57} C_VEL
LIN {X 0,Y 428.739,Z 534.019,A -85,B 0,C 180,E1 12410.74,E2 12410.74} C_VEL
LIN {X 0,Y 430.297,Z 536.444,A -85,B 0,C 180,E1 12407.042,E2 12407.042} C_VEL
LIN {X 0,Y 432.642,Z 540.976,A -85,B 0,C 180,E1 12403.968,E2 12403.968} C_VEL
LIN {X 0,Y 435.822,Z 546.85,A -85,B 0,C 180,E1 12401.056,E2 12401.056} C_VEL
LIN {X 0,Y 439.996,Z 555.142,A -85,B 0,C 180,E1 12398.083,E2 12398.083} C_VEL
LIN {X 0,Y 443.393,Z 562.13,A -85,B 0,C 180,E1 12396.056,E2 12396.056} C_VEL
LIN {X 0,Y 421.952,Z 792.502,A -85,B 0,C 180,E1 12392.621,E2 12392.621} C_VEL
LIN {X 0,Y 419.022,Z 814.841,A -85,B 0,C 180,E1 12392.229,E2 12392.229} C_VEL
LIN {X 0,Y 414.669,Z 839.207,A -85,B 0,C 180,E1 12391.69,E2 12391.69} C_VEL
LIN {X 0,Y 408.462,Z 865.63,A -85,B 0,C 180,E1 12390.913,E2 12390.913} C_VEL
LIN {X 0,Y 402.411,Z 886.895,A -85,B 0,C 180,E1 12390.129,E2 12390.129} C_VEL
LIN {X 0,Y 395.65,Z 907.39,A -85,B 0,C 180,E1 12389.229,E2 12389.229} C_VEL
LIN {X 0,Y 385.652,Z 933.455,A -85,B 0,C 180,E1 12387.832,E2 12387.832} C_VEL
LIN {X 0,Y 376.913,Z 953.302,A -85,B 0,C 180,E1 12386.542,E2 12386.542} C_VEL
LIN {X 0,Y 367.662,Z 972.354,A -85,B 0,C 180,E1 12385.078,E2 12385.078} C_VEL
LIN {X 0,Y 355.556,Z 994.846,A -85,B 0,C 180,E1 12383,E2 12383} C_VEL
LIN {X 0,Y 344.864,Z 1012.802,A -85,B 0,C 180,E1 12380.987,E2 12380.987} C_VEL
LIN {X 0,Y 334.583,Z 1028.894,A -85,B 0,C 180,E1 12378.857,E2 12378.857} C_VEL
LIN {X 0,Y 322.348,Z 1046.829,A -85,B 0,C 180,E1 12376.023,E2 12376.023} C_VEL
LIN {X 0,Y 310.839,Z 1062.438,A -85,B 0,C 180,E1 12372.994,E2 12372.994} C_VEL
LIN {X 0,Y 301.204,Z 1074.991,A -85,B 0,C 180,E1 12370.09,E2 12370.09} C_VEL
LIN {X 0,Y 290.422,Z 1088.634,A -85,B 0,C 180,E1 12366.31,E2 12366.31} C_VEL
LIN {X 0,Y 279.969,Z 1101.38,A -85,B 0,C 180,E1 12361.908,E2 12361.908} C_VEL
LIN {X 0,Y 272.034,Z 1111.039,A -85,B 0,C 180,E1 12357.826,E2 12357.826} C_VEL
LIN {X 0,Y 264.755,Z 1120.167,A -85,B 0,C 180,E1 12353.126,E2 12353.126} C_VEL
LIN {X 0,Y 258.059,Z 1128.938,A -85,B 0,C 180,E1 12347.358,E2 12347.358} C_VEL
LIN {X 0,Y 254.092,Z 1134.715,A -85,B 0,C 180,E1 12342.499,E2 12342.499} C_VEL
LIN {X 0,Y 251.486,Z 1139.15,A -85,B 0,C 180,E1 12337.769,E2 12337.769} C_VEL
LIN {X 0,Y 249.678,Z 1143.172,A -85,B 0,C 180,E1 12332.065,E2 12332.065} C_VEL
LIN {X 0,Y 248.932,Z 1145.568,A -85,B 0,C 180,E1 12326.546,E2 12326.546} C_VEL
LIN {X 0,Y 248.798,Z 1146.66,A -85,B 0,C 180,E1 12321.914,E2 12321.914} C_VEL
LIN {X 0,Y 248.913,Z 1146.9,A -85,B 0,C 180,E1 12317.236,E2 12317.236} C_VEL
LIN {X 0,Y 249.356,Z 1146.318,A -85,B 0,C 180,E1 12312.739,E2 12312.739} C_VEL
LIN {X 0,Y 250.445,Z 1144.81,A -85,B 0,C 180,E1 12307.958,E2 12307.958} C_VEL
LIN {X 0,Y 252.579,Z 1142.206,A -85,B 0,C 180,E1 12302.92,E2 12302.92} C_VEL
LIN {X 0,Y 256.994,Z 1137.467,A -85,B 0,C 180,E1 12296.731,E2 12296.731} C_VEL
LIN {X 0,Y 262.933,Z 1131.456,A -85,B 0,C 180,E1 12291.223,E2 12291.223} C_VEL
LIN {X 0,Y 269.632,Z 1125.023,A -85,B 0,C 180,E1 12286.622,E2 12286.622} C_VEL
LIN {X 0,Y 279.656,Z 1115.585,A -85,B 0,C 180,E1 12281.339,E2 12281.339} C_VEL
LIN {X 0,Y 290.204,Z 1105.385,A -85,B 0,C 180,E1 12276.934,E2 12276.934} C_VEL
LIN {X 0,Y 300.52,Z 1095.244,A -85,B 0,C 180,E1 12273.373,E2 12273.373} C_VEL
LIN {X 0,Y 313.747,Z 1081.818,A -85,B 0,C 180,E1 12269.541,E2 12269.541} C_VEL
LIN {X 0,Y 326.816,Z 1067.547,A -85,B 0,C 180,E1 12266.311,E2 12266.311} C_VEL
LIN {X 0,Y 337.949,Z 1054.756,A -85,B 0,C 180,E1 12263.906,E2 12263.906} C_VEL
LIN {X 0,Y 349.955,Z 1040.114,A -85,B 0,C 180,E1 12261.589,E2 12261.589} C_VEL
LIN {X 0,Y 364.915,Z 1020.356,A -85,B 0,C 180,E1 12259.03,E2 12259.03} C_VEL
LIN {X 0,Y 376.8,Z 1003.081,A -85,B 0,C 180,E1 12257.2,E2 12257.2} C_VEL
LIN {X 0,Y 387.398,Z 986.364,A -85,B 0,C 180,E1 12255.699,E2 12255.699} C_VEL
LIN {X 0,Y 399.52,Z 965.461,A -85,B 0,C 180,E1 12254.123,E2 12254.123} C_VEL
LIN {X 0,Y 411.037,Z 942.758,A -85,B 0,C 180,E1 12252.724,E2 12252.724} C_VEL
LIN {X 0,Y 419.719,Z 923.57,A -85,B 0,C 180,E1 12251.738,E2 12251.738} C_VEL
LIN {X 0,Y 427.619,Z 903.904,A -85,B 0,C 180,E1 12250.874,E2 12250.874} C_VEL
LIN {X 0,Y 432.537,Z 890.198,A -85,B 0,C 180,E1 12250.36,E2 12250.36} C_VEL
LIN {X 0,Y 434.713,Z 883.269,A -85,B 0,C 180,E1 12249.994,E2 12249.994} C_VEL
LIN {X 0,Y 438.761,Z 866.278,A -85,B 0,C 180,E1 12248.686,E2 12248.686} C_VEL
LIN {X 0,Y 440.487,Z 859.152,A -85,B 0,C 180,E1 12248.361,E2 12248.361} C_VEL
LIN {X 0,Y 445.816,Z 837.176,A -85,B 0,C 180,E1 12247.843,E2 12247.843} C_VEL
LIN {X 0,Y 450.031,Z 815.386,A -85,B 0,C 180,E1 12247.433,E2 12247.433} C_VEL
LIN {X 0,Y 453.786,Z 788.808,A -85,B 0,C 180,E1 12247.031,E2 12247.031} C_VEL
LIN {X 0,Y 474.89,Z 593.825,A -85,B 0,C 180,E1 12244.347,E2 12244.347} C_VEL
LIN {X 0,Y 473.457,Z 590.571,A -85,B 0,C 180,E1 12242.057,E2 12242.057} C_VEL
LIN {X 0,Y 472.42,Z 587.996,A -85,B 0,C 180,E1 12238.059,E2 12238.059} C_VEL
LIN {X 0,Y 472.606,Z 589,A -85,B 0,C 180,E1 12235.753,E2 12235.753} C_VEL
LIN {X 0,Y 473.743,Z 591.316,A -85,B 0,C 180,E1 12232.968,E2 12232.968} C_VEL
LIN {X 0,Y 475.288,Z 595.103,A -85,B 0,C 180,E1 12230.716,E2 12230.716} C_VEL
LIN {X 0,Y 452.428,Z 806.135,A -85,B 0,C 180,E1 12227.693,E2 12227.693} C_VEL
LIN {X 0,Y 448.851,Z 829.439,A -85,B 0,C 180,E1 12227.322,E2 12227.322} C_VEL
LIN {X 0,Y 442.41,Z 859.149,A -85,B 0,C 180,E1 12226.782,E2 12226.782} C_VEL
LIN {X 0,Y 436.362,Z 880.931,A -85,B 0,C 180,E1 12226.296,E2 12226.296} C_VEL
LIN {X 0,Y 429.558,Z 901.829,A -85,B 0,C 180,E1 12225.715,E2 12225.715} C_VEL
LIN {X 0,Y 420.477,Z 925.987,A -85,B 0,C 180,E1 12224.891,E2 12224.891} C_VEL
LIN {X 0,Y 409.754,Z 950.315,A -85,B 0,C 180,E1 12223.848,E2 12223.848} C_VEL
LIN {X 0,Y 399.823,Z 970.376,A -85,B 0,C 180,E1 12222.802,E2 12222.802} C_VEL
LIN {X 0,Y 389.755,Z 988.873,A -85,B 0,C 180,E1 12221.655,E2 12221.655} C_VEL
LIN {X 0,Y 376.619,Z 1010.961,A -85,B 0,C 180,E1 12220.02,E2 12220.02} C_VEL
LIN {X 0,Y 362.259,Z 1032.574,A -85,B 0,C 180,E1 12218.03,E2 12218.03} C_VEL
LIN {X 0,Y 349.929,Z 1049.805,A -85,B 0,C 180,E1 12216.112,E2 12216.112} C_VEL
LIN {X 0,Y 337.316,Z 1066.369,A -85,B 0,C 180,E1 12213.915,E2 12213.915} C_VEL
LIN {X 0,Y 321.123,Z 1086.248,A -85,B 0,C 180,E1 12210.671,E2 12210.671} C_VEL
LIN {X 0,Y 308.603,Z 1100.778,A -85,B 0,C 180,E1 12207.739,E2 12207.739} C_VEL
LIN {X 0,Y 296.952,Z 1113.867,A -85,B 0,C 180,E1 12204.571,E2 12204.571} C_VEL
LIN {X 0,Y 284.123,Z 1128.032,A -85,B 0,C 180,E1 12200.415,E2 12200.415} C_VEL
LIN {X 0,Y 271.933,Z 1141.287,A -85,B 0,C 180,E1 12195.505,E2 12195.505} C_VEL
LIN {X 0,Y 263.182,Z 1151.005,A -85,B 0,C 180,E1 12191.09,E2 12191.09} C_VEL
LIN {X 0,Y 255.824,Z 1159.59,A -85,B 0,C 180,E1 12186.375,E2 12186.375} C_VEL
LIN {X 0,Y 248.961,Z 1168.446,A -85,B 0,C 180,E1 12180.4,E2 12180.4} C_VEL
LIN {X 0,Y 244.189,Z 1175.597,A -85,B 0,C 180,E1 12174.058,E2 12174.058} C_VEL
LIN {X 0,Y 241.857,Z 1180.205,A -85,B 0,C 180,E1 12168.784,E2 12168.784} C_VEL
LIN {X 0,Y 240.778,Z 1183.421,A -85,B 0,C 180,E1 12163.937,E2 12163.937} C_VEL
LIN {X 0,Y 240.468,Z 1185.575,A -85,B 0,C 180,E1 12159.332,E2 12159.332} C_VEL
LIN {X 0,Y 240.531,Z 1186.78,A -85,B 0,C 180,E1 12155.008,E2 12155.008} C_VEL
LIN {X 0,Y 240.63,Z 1187.12,A -85,B 0,C 180,E1 12150.476,E2 12150.476} C_VEL
LIN {X 0,Y 240.588,Z 1186.485,A -85,B 0,C 180,E1 12145.949,E2 12145.949} C_VEL
LIN {X 0,Y 240.528,Z 1184.745,A -85,B 0,C 180,E1 12141.153,E2 12141.153} C_VEL
LIN {X 0,Y 240.82,Z 1181.921,A -85,B 0,C 180,E1 12136.307,E2 12136.307} C_VEL
LIN {X 0,Y 241.84,Z 1178.025,A -85,B 0,C 180,E1 12131.437,E2 12131.437} C_VEL
LIN {X 0,Y 243.853,Z 1173.036,A -85,B 0,C 180,E1 12126.564,E2 12126.564} C_VEL
LIN {X 0,Y 247.014,Z 1166.928,A -85,B 0,C 180,E1 12121.733,E2 12121.733} C_VEL
LIN {X 0,Y 251.677,Z 1159.28,A -85,B 0,C 180,E1 12116.754,E2 12116.754} C_VEL
LIN {X 0,Y 259.141,Z 1148.505,A -85,B 0,C 180,E1 12111.03,E2 12111.03} C_VEL
LIN {X 0,Y 267.825,Z 1136.618,A -85,B 0,C 180,E1 12106.022,E2 12106.022} C_VEL
LIN {X 0,Y 276.269,Z 1125.459,A -85,B 0,C 180,E1 12102.105,E2 12102.105} C_VEL
LIN {X 0,Y 285.8,Z 1112.939,A -85,B 0,C 180,E1 12098.404,E2 12098.404} C_VEL
LIN {X 0,Y 298.677,Z 1095.71,A -85,B 0,C 180,E1 12094.222,E2 12094.222} C_VEL
LIN {X 0,Y 309.723,Z 1080.367,A -85,B 0,C 180,E1 12091.187,E2 12091.187} C_VEL
LIN {X 0,Y 320.522,Z 1064.785,A -85,B 0,C 180,E1 12088.587,E2 12088.587} C_VEL
LIN {X 0,Y 333,Z 1045.863,A -85,B 0,C 180,E1 12085.938,E2 12085.938} C_VEL
LIN {X 0,Y 345.952,Z 1024.521,A -85,B 0,C 180,E1 12083.507,E2 12083.507} C_VEL
LIN {X 0,Y 356.337,Z 1006.097,A -85,B 0,C 180,E1 12081.758,E2 12081.758} C_VEL
LIN {X 0,Y 366.086,Z 987.436,A -85,B 0,C 180,E1 12080.254,E2 12080.254} C_VEL
LIN {X 0,Y 377.682,Z 962.944,A -85,B 0,C 180,E1 12078.603,E2 12078.603} C_VEL
LIN {X 0,Y 386.958,Z 940.734,A -85,B 0,C 180,E1 12077.39,E2 12077.39} C_VEL
LIN {X 0,Y 394.604,Z 920.258,A -85,B 0,C 180,E1 12076.454,E2 12076.454} C_VEL
LIN {X 0,Y 402.061,Z 897.649,A -85,B 0,C 180,E1 12075.598,E2 12075.598} C_VEL
LIN {X 0,Y 409.779,Z 869.561,A -85,B 0,C 180,E1 12074.761,E2 12074.761} C_VEL
LIN {X 0,Y 414.793,Z 847.067,A -85,B 0,C 180,E1 12074.244,E2 12074.244} C_VEL
LIN {X 0,Y 418.734,Z 824.352,A -85,B 0,C 180,E1 12073.798,E2 12073.798} C_VEL
LIN {X 0,Y 422.31,Z 793.717,A -85,B 0,C 180,E1 12073.285,E2 12073.285} C_VEL
LIN {X 0,Y 442.805,Z 572.2,A -85,B 0,C 180,E1 12069.927,E2 12069.927} C_VEL
LIN {X 0,Y 439.346,Z 564.708,A -85,B 0,C 180,E1 12067.881,E2 12067.881} C_VEL
LIN {X 0,Y 435.575,Z 557.124,A -85,B 0,C 180,E1 12065.268,E2 12065.268} C_VEL
LIN {X 0,Y 432.756,Z 551.325,A -85,B 0,C 180,E1 12062.847,E2 12062.847} C_VEL
LIN {X 0,Y 430.717,Z 547.491,A -85,B 0,C 180,E1 12060.665,E2 12060.665} C_VEL
LIN {X 0,Y 428.881,Z 543.771,A -85,B 0,C 180,E1 12057.862,E2 12057.862} C_VEL
LIN {X 0,Y 427.572,Z 541.442,A -85,B 0,C 180,E1 12053.42,E2 12053.42} C_VEL
LIN {X 0,Y 427.792,Z 542.047,A -85,B 0,C 180,E1 12050.583,E2 12050.583} C_VEL
LIN {X 0,Y 429.24,Z 544.373,A -85,B 0,C 180,E1 12047.146,E2 12047.146} C_VEL
LIN {X 0,Y 431.483,Z 548.824,A -85,B 0,C 180,E1 12044.131,E2 12044.131} C_VEL
LIN {X 0,Y 434.436,Z 554.432,A -85,B 0,C 180,E1 12041.342,E2 12041.342} C_VEL
LIN {X 0,Y 438.454,Z 562.65,A -85,B 0,C 180,E1 12038.389,E2 12038.389} C_VEL
LIN {X 0,Y 440.683,Z 567.536,A -85,B 0,C 180,E1 12036.976,E2 12036.976} C_VEL
LIN {X 0,Y 419.071,Z 794.57,A -85,B 0,C 180,E1 12033.619,E2 12033.619} C_VEL
LIN {X 0,Y 416.041,Z 816.784,A -85,B 0,C 180,E1 12033.229,E2 12033.229} C_VEL
LIN {X 0,Y 411.062,Z 843.42,A -85,B 0,C 180,E1 12032.63,E2 12032.63} C_VEL
LIN {X 0,Y 405.152,Z 867.457,A -85,B 0,C 180,E1 12031.916,E2 12031.916} C_VEL
LIN {X 0,Y 399.388,Z 887.32,A -85,B 0,C 180,E1 12031.189,E2 12031.189} C_VEL
LIN {X 0,Y 392.504,Z 907.838,A -85,B 0,C 180,E1 12030.303,E2 12030.303} C_VEL
LIN {X 0,Y 382.32,Z 933.918,A -85,B 0,C 180,E1 12028.924,E2 12028.924} C_VEL
LIN {X 0,Y 373.411,Z 953.771,A -85,B 0,C 180,E1 12027.649,E2 12027.649} C_VEL
LIN {X 0,Y 364.332,Z 972.127,A -85,B 0,C 180,E1 12026.257,E2 12026.257} C_VEL
LIN {X 0,Y 352.653,Z 993.589,A -85,B 0,C 180,E1 12024.321,E2 12024.321} C_VEL
LIN {X 0,Y 340.94,Z 1012.858,A -85,B 0,C 180,E1 12022.197,E2 12022.197} C_VEL
LIN {X 0,Y 330.758,Z 1028.448,A -85,B 0,C 180,E1 12020.159,E2 12020.159} C_VEL
LIN {X 0,Y 319.38,Z 1044.783,A -85,B 0,C 180,E1 12017.631,E2 12017.631} C_VEL
LIN {X 0,Y 306.256,Z 1062.246,A -85,B 0,C 180,E1 12014.32,E2 12014.32} C_VEL
LIN {X 0,Y 295.723,Z 1075.544,A -85,B 0,C 180,E1 12011.247,E2 12011.247} C_VEL
LIN {X 0,Y 285.026,Z 1088.601,A -85,B 0,C 180,E1 12007.617,E2 12007.617} C_VEL
LIN {X 0,Y 273.675,Z 1101.957,A -85,B 0,C 180,E1 12002.981,E2 12002.981} C_VEL
LIN {X 0,Y 265.389,Z 1111.622,A -85,B 0,C 180,E1 11998.832,E2 11998.832} C_VEL
LIN {X 0,Y 257.751,Z 1120.762,A -85,B 0,C 180,E1 11994.036,E2 11994.036} C_VEL
LIN {X 0,Y 250.692,Z 1129.548,A -85,B 0,C 180,E1 11988.125,E2 11988.125} C_VEL
LIN {X 0,Y 246.486,Z 1135.33,A -85,B 0,C 180,E1 11983.13,E2 11983.13} C_VEL
LIN {X 0,Y 243.707,Z 1139.771,A -85,B 0,C 180,E1 11978.256,E2 11978.256} C_VEL
LIN {X 0,Y 241.767,Z 1143.799,A -85,B 0,C 180,E1 11972.37,E2 11972.37} C_VEL
LIN {X 0,Y 240.968,Z 1146.21,A -85,B 0,C 180,E1 11966.67,E2 11966.67} C_VEL
LIN {X 0,Y 240.823,Z 1147.313,A -85,B 0,C 180,E1 11961.885,E2 11961.885} C_VEL
LIN {X 0,Y 240.95,Z 1147.565,A -85,B 0,C 180,E1 11957.051,E2 11957.051} C_VEL
LIN {X 0,Y 241.463,Z 1146.966,A -85,B 0,C 180,E1 11952.256,E2 11952.256} C_VEL
LIN {X 0,Y 242.657,Z 1145.471,A -85,B 0,C 180,E1 11947.371,E2 11947.371} C_VEL
LIN {X 0,Y 244.935,Z 1142.92,A -85,B 0,C 180,E1 11942.266,E2 11942.266} C_VEL
LIN {X 0,Y 249.669,Z 1138.211,A -85,B 0,C 180,E1 11935.898,E2 11935.898} C_VEL
LIN {X 0,Y 255.865,Z 1132.325,A -85,B 0,C 180,E1 11930.341,E2 11930.341} C_VEL
LIN {X 0,Y 262.974,Z 1125.872,A -85,B 0,C 180,E1 11925.606,E2 11925.606} C_VEL
LIN {X 0,Y 273.149,Z 1116.808,A -85,B 0,C 180,E1 11920.386,E2 11920.386} C_VEL
LIN {X 0,Y 284.574,Z 1106.221,A -85,B 0,C 180,E1 11915.745,E2 11915.745} C_VEL
LIN {X 0,Y 295.542,Z 1095.857,A -85,B 0,C 180,E1 11912.085,E2 11912.085} C_VEL
LIN {X 0,Y 308.958,Z 1082.725,A -85,B 0,C 180,E1 11908.327,E2 11908.327} C_VEL
LIN {X 0,Y 323.113,Z 1067.723,A -85,B 0,C 180,E1 11904.95,E2 11904.95} C_VEL
LIN {X 0,Y 335.32,Z 1054.053,A -85,B 0,C 180,E1 11902.428,E2 11902.428} C_VEL
LIN {X 0,Y 349.661,Z 1036.919,A -85,B 0,C 180,E1 11899.817,E2 11899.817} C_VEL
LIN {X 0,Y 363.83,Z 1018.143,A -85,B 0,C 180,E1 11897.521,E2 11897.521} C_VEL
LIN {X 0,Y 374.772,Z 1002.469,A -85,B 0,C 180,E1 11895.919,E2 11895.919} C_VEL
LIN {X 0,Y 386.062,Z 984.895,A -85,B 0,C 180,E1 11894.391,E2 11894.391} C_VEL
LIN {X 0,Y 399.717,Z 961.172,A -85,B 0,C 180,E1 11892.695,E2 11892.695} C_VEL
LIN {X 0,Y 409.648,Z 941.653,A -85,B 0,C 180,E1 11891.546,E2 11891.546} C_VEL
LIN {X 0,Y 418.512,Z 922.232,A -85,B 0,C 180,E1 11890.584,E2 11890.584} C_VEL
LIN {X 0,Y 427.944,Z 898.788,A -85,B 0,C 180,E1 11889.609,E2 11889.609} C_VEL
LIN {X 0,Y 436.057,Z 874.403,A -85,B 0,C 180,E1 11888.787,E2 11888.787} C_VEL
LIN {X 0,Y 440.487,Z 859.152,A -85,B 0,C 180,E1 11888.361,E2 11888.361} C_VEL
LIN {X 0,Y 442.163,Z 851.947,A -85,B 0,C 180,E1 11888.05,E2 11888.05} C_VEL
LIN {X 0,Y 445.534,Z 833.226,A -85,B 0,C 180,E1 11886.839,E2 11886.839} C_VEL
LIN {X 0,Y 446.72,Z 826.921,A -85,B 0,C 180,E1 11886.622,E2 11886.622} C_VEL
LIN {X 0,Y 450.993,Z 800.58,A -85,B 0,C 180,E1 11886.196,E2 11886.196} C_VEL
LIN {X 0,Y 473.259,Z 600.563,A -85,B 0,C 180,E1 11883.467,E2 11883.467} C_VEL
LIN {X 0,Y 472.412,Z 598.45,A -85,B 0,C 180,E1 11881.941,E2 11881.941} C_VEL
LIN {X 0,Y 471.438,Z 595.937,A -85,B 0,C 180,E1 11878.055,E2 11878.055} C_VEL
LIN {X 0,Y 471.598,Z 596.886,A -85,B 0,C 180,E1 11875.866,E2 11875.866} C_VEL
LIN {X 0,Y 472.684,Z 599.222,A -85,B 0,C 180,E1 11873.075,E2 11873.075} C_VEL
LIN {X 0,Y 473.593,Z 601.743,A -85,B 0,C 180,E1 11871.586,E2 11871.586} C_VEL
LIN {X 0,Y 450.99,Z 806.478,A -85,B 0,C 180,E1 11868.691,E2 11868.691} C_VEL
LIN {X 0,Y 447.123,Z 830.964,A -85,B 0,C 180,E1 11868.307,E2 11868.307} C_VEL
LIN {X 0,Y 440.797,Z 859.284,A -85,B 0,C 180,E1 11867.802,E2 11867.802} C_VEL
LIN {X 0,Y 434.764,Z 880.708,A -85,B 0,C 180,E1 11867.338,E2 11867.338} C_VEL
LIN {X 0,Y 427.797,Z 901.798,A -85,B 0,C 180,E1 11866.769,E2 11866.769} C_VEL
LIN {X 0,Y 418.452,Z 926.271,A -85,B 0,C 180,E1 11865.955,E2 11865.955} C_VEL
LIN {X 0,Y 407.894,Z 949.785,A -85,B 0,C 180,E1 11864.972,E2 11864.972} C_VEL
LIN {X 0,Y 398.356,Z 968.815,A -85,B 0,C 180,E1 11864.011,E2 11864.011} C_VEL
LIN {X 0,Y 388.104,Z 987.406,A -85,B 0,C 180,E1 11862.9,E2 11862.9} C_VEL
LIN {X 0,Y 376.368,Z 1006.873,A -85,B 0,C 180,E1 11861.515,E2 11861.515} C_VEL
LIN {X 0,Y 360.855,Z 1030.172,A -85,B 0,C 180,E1 11859.477,E2 11859.477} C_VEL
LIN {X 0,Y 348.205,Z 1047.553,A -85,B 0,C 180,E1 11857.61,E2 11857.61} C_VEL
LIN {X 0,Y 336.338,Z 1062.827,A -85,B 0,C 180,E1 11855.666,E2 11855.666} C_VEL
LIN {X 0,Y 322.751,Z 1079.346,A -85,B 0,C 180,E1 11853.151,E2 11853.151} C_VEL
LIN {X 0,Y 306.17,Z 1098.263,A -85,B 0,C 180,E1 11849.558,E2 11849.558} C_VEL
LIN {X 0,Y 293.972,Z 1111.511,A -85,B 0,C 180,E1 11846.439,E2 11846.439} C_VEL
LIN {X 0,Y 282.558,Z 1123.592,A -85,B 0,C 180,E1 11843.017,E2 11843.017} C_VEL
LIN {X 0,Y 270.914,Z 1135.764,A -85,B 0,C 180,E1 11838.842,E2 11838.842} C_VEL
LIN {X 0,Y 258.486,Z 1148.78,A -85,B 0,C 180,E1 11833.209,E2 11833.209} C_VEL
LIN {X 0,Y 250.146,Z 1157.827,A -85,B 0,C 180,E1 11828.283,E2 11828.283} C_VEL
LIN {X 0,Y 243.766,Z 1165.265,A -85,B 0,C 180,E1 11823.342,E2 11823.342} C_VEL
LIN {X 0,Y 238.533,Z 1172.125,A -85,B 0,C 180,E1 11817.728,E2 11817.728} C_VEL
LIN {X 0,Y 234.516,Z 1178.662,A -85,B 0,C 180,E1 11810.724,E2 11810.724} C_VEL
LIN {X 0,Y 232.938,Z 1182.531,A -85,B 0,C 180,E1 11804.924,E2 11804.924} C_VEL
LIN {X 0,Y 232.498,Z 1184.855,A -85,B 0,C 180,E1 11799.905,E2 11799.905} C_VEL
LIN {X 0,Y 232.548,Z 1186.128,A -85,B 0,C 180,E1 11795.181,E2 11795.181} C_VEL
LIN {X 0,Y 232.656,Z 1186.468,A -85,B 0,C 180,E1 11790.739,E2 11790.739} C_VEL
LIN {X 0,Y 232.616,Z 1185.863,A -85,B 0,C 180,E1 11786.057,E2 11786.057} C_VEL
LIN {X 0,Y 232.549,Z 1184.146,A -85,B 0,C 180,E1 11781.096,E2 11781.096} C_VEL
LIN {X 0,Y 232.895,Z 1181.169,A -85,B 0,C 180,E1 11775.835,E2 11775.835} C_VEL
LIN {X 0,Y 234.044,Z 1177.209,A -85,B 0,C 180,E1 11770.764,E2 11770.764} C_VEL
LIN {X 0,Y 236.221,Z 1172.209,A -85,B 0,C 180,E1 11765.759,E2 11765.759} C_VEL
LIN {X 0,Y 239.734,Z 1165.899,A -85,B 0,C 180,E1 11760.658,E2 11760.658} C_VEL
LIN {X 0,Y 244.911,Z 1157.992,A -85,B 0,C 180,E1 11755.426,E2 11755.426} C_VEL
LIN {X 0,Y 253.657,Z 1146.024,A -85,B 0,C 180,E1 11749.131,E2 11749.131} C_VEL
LIN {X 0,Y 261.952,Z 1135.32,A -85,B 0,C 180,E1 11744.616,E2 11744.616} C_VEL
LIN {X 0,Y 271.074,Z 1123.77,A -85,B 0,C 180,E1 11740.551,E2 11740.551} C_VEL
LIN {X 0,Y 283.321,Z 1108.32,A -85,B 0,C 180,E1 11736.084,E2 11736.084} C_VEL
LIN {X 0,Y 295.162,Z 1092.834,A -85,B 0,C 180,E1 11732.49,E2 11732.49} C_VEL
LIN {X 0,Y 306.025,Z 1078.184,A -85,B 0,C 180,E1 11729.648,E2 11729.648} C_VEL
LIN {X 0,Y 317.558,Z 1061.938,A -85,B 0,C 180,E1 11726.995,E2 11726.995} C_VEL
LIN {X 0,Y 331.918,Z 1040.351,A -85,B 0,C 180,E1 11724.113,E2 11724.113} C_VEL
LIN {X 0,Y 343.179,Z 1022.023,A -85,B 0,C 180,E1 11722.105,E2 11722.105} C_VEL
LIN {X 0,Y 353.467,Z 1004.04,A -85,B 0,C 180,E1 11720.44,E2 11720.44} C_VEL
LIN {X 0,Y 365.583,Z 981.078,A -85,B 0,C 180,E1 11718.663,E2 11718.663} C_VEL
LIN {X 0,Y 376.306,Z 958.015,A -85,B 0,C 180,E1 11717.215,E2 11717.215} C_VEL
LIN {X 0,Y 384.708,Z 937.999,A -85,B 0,C 180,E1 11716.166,E2 11716.166} C_VEL
LIN {X 0,Y 392.733,Z 916.597,A -85,B 0,C 180,E1 11715.227,E2 11715.227} C_VEL
LIN {X 0,Y 401.783,Z 888.345,A -85,B 0,C 180,E1 11714.237,E2 11714.237} C_VEL
LIN {X 0,Y 407.771,Z 865.828,A -85,B 0,C 180,E1 11713.621,E2 11713.621} C_VEL
LIN {X 0,Y 412.659,Z 843.623,A -85,B 0,C 180,E1 11713.133,E2 11713.133} C_VEL
LIN {X 0,Y 417.219,Z 815.971,A -85,B 0,C 180,E1 11712.612,E2 11712.612} C_VEL
LIN {X 0,Y 422.137,Z 766.914,A -85,B 0,C 180,E1 11711.848,E2 11711.848} C_VEL
LIN {X 0,Y 440.06,Z 577.146,A -85,B 0,C 180,E1 11708.987,E2 11708.987} C_VEL
LIN {X 0,Y 436.214,Z 568.892,A -85,B 0,C 180,E1 11706.515,E2 11706.515} C_VEL
LIN {X 0,Y 432.434,Z 561.04,A -85,B 0,C 180,E1 11703.513,E2 11703.513} C_VEL
LIN {X 0,Y 429.83,Z 555.695,A -85,B 0,C 180,E1 11700.8,E2 11700.8} C_VEL
LIN {X 0,Y 427.817,Z 551.642,A -85,B 0,C 180,E1 11697.723,E2 11697.723} C_VEL
LIN {X 0,Y 426.592,Z 549.381,A -85,B 0,C 180,E1 11693.405,E2 11693.405} C_VEL
LIN {X 0,Y 426.788,Z 549.947,A -85,B 0,C 180,E1 11690.697,E2 11690.697} C_VEL
LIN {X 0,Y 428.15,Z 552.197,A -85,B 0,C 180,E1 11687.319,E2 11687.319} C_VEL
LIN {X 0,Y 430.271,Z 556.54,A -85,B 0,C 180,E1 11684.361,E2 11684.361} C_VEL
LIN {X 0,Y 433.135,Z 562.192,A -85,B 0,C 180,E1 11681.563,E2 11681.563} C_VEL
LIN {X 0,Y 436.925,Z 570.157,A -85,B 0,C 180,E1 11678.697,E2 11678.697} C_VEL
LIN {X 0,Y 438.086,Z 572.933,A -85,B 0,C 180,E1 11677.909,E2 11677.909} C_VEL
LIN {X 0,Y 416.383,Z 796.091,A -85,B 0,C 180,E1 11674.64,E2 11674.64} C_VEL
LIN {X 0,Y 413.139,Z 819.036,A -85,B 0,C 180,E1 11674.236,E2 11674.236} C_VEL
LIN {X 0,Y 407.549,Z 847.262,A -85,B 0,C 180,E1 11673.588,E2 11673.588} C_VEL
LIN {X 0,Y 401.968,Z 869.277,A -85,B 0,C 180,E1 11672.935,E2 11672.935} C_VEL
LIN {X 0,Y 395.717,Z 890.193,A -85,B 0,C 180,E1 11672.171,E2 11672.171} C_VEL
LIN {X 0,Y 387.195,Z 914.596,A -85,B 0,C 180,E1 11671.093,E2 11671.093} C_VEL
LIN {X 0,Y 377.987,Z 936.944,A -85,B 0,C 180,E1 11669.881,E2 11669.881} C_VEL
LIN {X 0,Y 369.476,Z 955.429,A -85,B 0,C 180,E1 11668.695,E2 11668.695} C_VEL
LIN {X 0,Y 359.325,Z 975.414,A -85,B 0,C 180,E1 11667.176,E2 11667.176} C_VEL
LIN {X 0,Y 346.711,Z 997.565,A -85,B 0,C 180,E1 11665.13,E2 11665.13} C_VEL
LIN {X 0,Y 336.239,Z 1014.332,A -85,B 0,C 180,E1 11663.264,E2 11663.264} C_VEL
LIN {X 0,Y 325.777,Z 1029.92,A -85,B 0,C 180,E1 11661.22,E2 11661.22} C_VEL
LIN {X 0,Y 312.863,Z 1047.888,A -85,B 0,C 180,E1 11658.402,E2 11658.402} C_VEL
LIN {X 0,Y 300.651,Z 1063.516,A -85,B 0,C 180,E1 11655.372,E2 11655.372} C_VEL
LIN {X 0,Y 289.816,Z 1076.754,A -85,B 0,C 180,E1 11652.279,E2 11652.279} C_VEL
LIN {X 0,Y 277.795,Z 1090.943,A -85,B 0,C 180,E1 11648.248,E2 11648.248} C_VEL
LIN {X 0,Y 266.606,Z 1103.504,A -85,B 0,C 180,E1 11643.714,E2 11643.714} C_VEL
LIN {X 0,Y 258.449,Z 1112.639,A -85,B 0,C 180,E1 11639.682,E2 11639.682} C_VEL
LIN {X 0,Y 249.889,Z 1122.491,A -85,B 0,C 180,E1 11634.338,E2 11634.338} C_VEL
LIN {X 0,Y 243.135,Z 1130.437,A -85,B 0,C 180,E1 11628.709,E2 11628.709} C_VEL
LIN {X 0,Y 238.74,Z 1136.182,A -85,B 0,C 180,E1 11623.564,E2 11623.564} C_VEL
LIN {X 0,Y 235.618,Z 1140.971,A -85,B 0,C 180,E1 11618.05,E2 11618.05} C_VEL
LIN {X 0,Y 233.649,Z 1144.885,A -85,B 0,C 180,E1 11611.716,E2 11611.716} C_VEL
LIN {X 0,Y 232.967,Z 1146.984,A -85,B 0,C 180,E1 11606.309,E2 11606.309} C_VEL
LIN {X 0,Y 232.845,Z 1147.992,A -85,B 0,C 180,E1 11601.605,E2 11601.605} C_VEL
LIN {X 0,Y 232.988,Z 1148.232,A -85,B 0,C 180,E1 11596.853,E2 11596.853} C_VEL
LIN {X 0,Y 233.557,Z 1147.646,A -85,B 0,C 180,E1 11591.882,E2 11591.882} C_VEL
LIN {X 0,Y 234.84,Z 1146.184,A -85,B 0,C 180,E1 11586.879,E2 11586.879} C_VEL
LIN {X 0,Y 237.322,Z 1143.635,A -85,B 0,C 180,E1 11581.57,E2 11581.57} C_VEL
LIN {X 0,Y 242.179,Z 1139.176,A -85,B 0,C 180,E1 11575.247,E2 11575.247} C_VEL
LIN {X 0,Y 248.877,Z 1133.178,A -85,B 0,C 180,E1 11569.396,E2 11569.396} C_VEL
LIN {X 0,Y 256.49,Z 1126.652,A -85,B 0,C 180,E1 11564.49,E2 11564.49} C_VEL
LIN {X 0,Y 267.114,Z 1117.657,A -85,B 0,C 180,E1 11559.209,E2 11559.209} C_VEL
LIN {X 0,Y 279.211,Z 1106.935,A -85,B 0,C 180,E1 11554.459,E2 11554.459} C_VEL
LIN {X 0,Y 290.294,Z 1096.864,A -85,B 0,C 180,E1 11550.878,E2 11550.878} C_VEL
LIN {X 0,Y 304.31,Z 1083.621,A -85,B 0,C 180,E1 11547.075,E2 11547.075} C_VEL
LIN {X 0,Y 318.882,Z 1068.676,A -85,B 0,C 180,E1 11543.713,E2 11543.713} C_VEL
LIN {X 0,Y 331.288,Z 1055.175,A -85,B 0,C 180,E1 11541.234,E2 11541.234} C_VEL
LIN {X 0,Y 344.51,Z 1039.8,A -85,B 0,C 180,E1 11538.891,E2 11538.891} C_VEL
LIN {X 0,Y 359.923,Z 1020.126,A -85,B 0,C 180,E1 11536.461,E2 11536.461} C_VEL
LIN {X 0,Y 371.546,Z 1003.881,A -85,B 0,C 180,E1 11534.813,E2 11534.813} C_VEL
LIN {X 0,Y 382.777,Z 986.795,A -85,B 0,C 180,E1 11533.341,E2 11533.341} C_VEL
LIN {X 0,Y 395.736,Z 965.118,A -85,B 0,C 180,E1 11531.785,E2 11531.785} C_VEL
LIN {X 0,Y 407.296,Z 942.922,A -85,B 0,C 180,E1 11530.486,E2 11530.486} C_VEL
LIN {X 0,Y 416.064,Z 924.104,A -85,B 0,C 180,E1 11529.569,E2 11529.569} C_VEL
LIN {X 0,Y 424.359,Z 904.019,A -85,B 0,C 180,E1 11528.732,E2 11528.732} C_VEL
LIN {X 0,Y 433.801,Z 877.103,A -85,B 0,C 180,E1 11527.816,E2 11527.816} C_VEL
LIN {X 0,Y 440.233,Z 854.758,A -85,B 0,C 180,E1 11527.212,E2 11527.212} C_VEL
LIN {X 0,Y 445.105,Z 834.309,A -85,B 0,C 180,E1 11526.765,E2 11526.765} C_VEL
LIN {X 0,Y 446.72,Z 826.921,A -85,B 0,C 180,E1 11526.622,E2 11526.622} C_VEL
LIN {X 0,Y 447.974,Z 819.521,A -85,B 0,C 180,E1 11526.366,E2 11526.366} C_VEL
LIN {X 0,Y 450.009,Z 800.188,A -85,B 0,C 180,E1 11525.277,E2 11525.277} C_VEL
LIN {X 0,Y 450.756,Z 793.747,A -85,B 0,C 180,E1 11525.088,E2 11525.088} C_VEL
LIN {X 0,Y 471.753,Z 607.256,A -85,B 0,C 180,E1 11522.589,E2 11522.589} C_VEL
LIN {X 0,Y 471.041,Z 605.775,A -85,B 0,C 180,E1 11521.095,E2 11521.095} C_VEL
LIN {X 0,Y 470.456,Z 603.862,A -85,B 0,C 180,E1 11517.929,E2 11517.929} C_VEL
LIN {X 0,Y 470.759,Z 605.306,A -85,B 0,C 180,E1 11515.248,E2 11515.248} C_VEL
LIN {X 0,Y 471.626,Z 607.127,A -85,B 0,C 180,E1 11513.181,E2 11513.181} C_VEL
LIN {X 0,Y 471.998,Z 608.461,A -85,B 0,C 180,E1 11512.462,E2 11512.462} C_VEL
LIN {X 0,Y 449.665,Z 807.19,A -85,B 0,C 180,E1 11509.691,E2 11509.691} C_VEL
LIN {X 0,Y 445.22,Z 834.242,A -85,B 0,C 180,E1 11509.272,E2 11509.272} C_VEL
LIN {X 0,Y 439.01,Z 860.623,A -85,B 0,C 180,E1 11508.806,E2 11508.806} C_VEL
LIN {X 0,Y 432.854,Z 881.954,A -85,B 0,C 180,E1 11508.352,E2 11508.352} C_VEL
LIN {X 0,Y 425.13,Z 904.735,A -85,B 0,C 180,E1 11507.744,E2 11507.744} C_VEL
LIN {X 0,Y 414.324,Z 931.546,A -85,B 0,C 180,E1 11506.84,E2 11506.84} C_VEL
LIN {X 0,Y 404.985,Z 951.71,A -85,B 0,C 180,E1 11505.994,E2 11505.994} C_VEL
LIN {X 0,Y 394.927,Z 971.233,A -85,B 0,C 180,E1 11505.014,E2 11505.014} C_VEL
LIN {X 0,Y 382.784,Z 992.571,A -85,B 0,C 180,E1 11503.727,E2 11503.727} C_VEL
LIN {X 0,Y 368.326,Z 1015.182,A -85,B 0,C 180,E1 11502.044,E2 11502.044} C_VEL
LIN {X 0,Y 355.992,Z 1032.829,A -85,B 0,C 180,E1 11500.442,E2 11500.442} C_VEL
LIN {X 0,Y 343.139,Z 1049.927,A -85,B 0,C 180,E1 11498.588,E2 11498.588} C_VEL
LIN {X 0,Y 327.594,Z 1069.212,A -85,B 0,C 180,E1 11496.049,E2 11496.049} C_VEL
LIN {X 0,Y 312.281,Z 1086.664,A -85,B 0,C 180,E1 11493.162,E2 11493.162} C_VEL
LIN {X 0,Y 299.685,Z 1100.347,A -85,B 0,C 180,E1 11490.409,E2 11490.409} C_VEL
LIN {X 0,Y 287.468,Z 1113.104,A -85,B 0,C 180,E1 11487.322,E2 11487.322} C_VEL
LIN {X 0,Y 273.053,Z 1127.772,A -85,B 0,C 180,E1 11482.965,E2 11482.965} C_VEL
LIN {X 0,Y 260.285,Z 1140.345,A -85,B 0,C 180,E1 11478.179,E2 11478.179} C_VEL
LIN {X 0,Y 250.639,Z 1150.011,A -85,B 0,C 180,E1 11473.641,E2 11473.641} C_VEL
LIN {X 0,Y 242.131,Z 1158.825,A -85,B 0,C 180,E1 11468.575,E2 11468.575} C_VEL
LIN {X 0,Y 233.833,Z 1168.193,A -85,B 0,C 180,E1 11461.732,E2 11461.732} C_VEL
LIN {X 0,Y 228.958,Z 1174.551,A -85,B 0,C 180,E1 11455.616,E2 11455.616} C_VEL
LIN {X 0,Y 226.275,Z 1178.974,A -85,B 0,C 180,E1 11450.161,E2 11450.161} C_VEL
LIN {X 0,Y 224.942,Z 1182.179,A -85,B 0,C 180,E1 11444.94,E2 11444.94} C_VEL
LIN {X 0,Y 224.517,Z 1184.304,A -85,B 0,C 180,E1 11440.002,E2 11440.002} C_VEL
LIN {X 0,Y 224.565,Z 1185.477,A -85,B 0,C 180,E1 11435.365,E2 11435.365} C_VEL
LIN {X 0,Y 224.684,Z 1185.799,A -85,B 0,C 180,E1 11430.765,E2 11430.765} C_VEL
LIN {X 0,Y 224.644,Z 1185.241,A -85,B 0,C 180,E1 11426.172,E2 11426.172} C_VEL
LIN {X 0,Y 224.57,Z 1183.547,A -85,B 0,C 180,E1 11421.035,E2 11421.035} C_VEL
LIN {X 0,Y 224.94,Z 1180.588,A -85,B 0,C 180,E1 11415.587,E2 11415.587} C_VEL
LIN {X 0,Y 226.16,Z 1176.65,A -85,B 0,C 180,E1 11410.341,E2 11410.341} C_VEL
LIN {X 0,Y 228.484,Z 1171.662,A -85,B 0,C 180,E1 11405.159,E2 11405.159} C_VEL
LIN {X 0,Y 232.147,Z 1165.465,A -85,B 0,C 180,E1 11399.967,E2 11399.967} C_VEL
LIN {X 0,Y 237.391,Z 1157.863,A -85,B 0,C 180,E1 11394.759,E2 11394.759} C_VEL
LIN {X 0,Y 245.724,Z 1147.04,A -85,B 0,C 180,E1 11388.763,E2 11388.763} C_VEL
LIN {X 0,Y 255.329,Z 1135.116,A -85,B 0,C 180,E1 11383.57,E2 11383.57} C_VEL
LIN {X 0,Y 264.53,Z 1123.935,A -85,B 0,C 180,E1 11379.55,E2 11379.55} C_VEL
LIN {X 0,Y 276.01,Z 1110.01,A -85,B 0,C 180,E1 11375.406,E2 11375.406} C_VEL
LIN {X 0,Y 289.358,Z 1093.262,A -85,B 0,C 180,E1 11371.407,E2 11371.407} C_VEL
LIN {X 0,Y 300.51,Z 1078.704,A -85,B 0,C 180,E1 11368.553,E2 11368.553} C_VEL
LIN {X 0,Y 311.609,Z 1063.554,A -85,B 0,C 180,E1 11366.047,E2 11366.047} C_VEL
LIN {X 0,Y 324.354,Z 1045.214,A -85,B 0,C 180,E1 11363.51,E2 11363.51} C_VEL
LIN {X 0,Y 338.105,Z 1023.655,A -85,B 0,C 180,E1 11361.092,E2 11361.092} C_VEL
LIN {X 0,Y 348.769,Z 1005.545,A -85,B 0,C 180,E1 11359.407,E2 11359.407} C_VEL
LIN {X 0,Y 358.913,Z 986.939,A -85,B 0,C 180,E1 11357.946,E2 11357.946} C_VEL
LIN {X 0,Y 370.525,Z 963.52,A -85,B 0,C 180,E1 11356.401,E2 11356.401} C_VEL
LIN {X 0,Y 380.751,Z 939.906,A -85,B 0,C 180,E1 11355.15,E2 11355.15} C_VEL
LIN {X 0,Y 388.436,Z 920.027,A -85,B 0,C 180,E1 11354.273,E2 11354.273} C_VEL
LIN {X 0,Y 395.85,Z 898.34,A -85,B 0,C 180,E1 11353.48,E2 11353.48} C_VEL
LIN {X 0,Y 403.938,Z 870.184,A -85,B 0,C 180,E1 11352.663,E2 11352.663} C_VEL
LIN {X 0,Y 409.329,Z 846.807,A -85,B 0,C 180,E1 11352.145,E2 11352.145} C_VEL
LIN {X 0,Y 413.34,Z 824.499,A -85,B 0,C 180,E1 11351.719,E2 11351.719} C_VEL
LIN {X 0,Y 416.862,Z 796.452,A -85,B 0,C 180,E1 11351.253,E2 11351.253} C_VEL
LIN {X 0,Y 437.458,Z 582.392,A -85,B 0,C 180,E1 11348.066,E2 11348.066} C_VEL
LIN {X 0,Y 433.427,Z 573.581,A -85,B 0,C 180,E1 11345.228,E2 11345.228} C_VEL
LIN {X 0,Y 430.183,Z 566.643,A -85,B 0,C 180,E1 11342.331,E2 11342.331} C_VEL
LIN {X 0,Y 428.39,Z 563.047,A -85,B 0,C 180,E1 11340.267,E2 11340.267} C_VEL
LIN {X 0,Y 426.755,Z 559.514,A -85,B 0,C 180,E1 11337.583,E2 11337.583} C_VEL
LIN {X 0,Y 425.611,Z 557.32,A -85,B 0,C 180,E1 11333.39,E2 11333.39} C_VEL
LIN {X 0,Y 425.813,Z 557.914,A -85,B 0,C 180,E1 11330.675,E2 11330.675} C_VEL
LIN {X 0,Y 427.098,Z 560.124,A -85,B 0,C 180,E1 11327.424,E2 11327.424} C_VEL
LIN {X 0,Y 429.12,Z 564.386,A -85,B 0,C 180,E1 11324.526,E2 11324.526} C_VEL
LIN {X 0,Y 431.769,Z 569.772,A -85,B 0,C 180,E1 11321.852,E2 11321.852} C_VEL
LIN {X 0,Y 435.407,Z 577.664,A -85,B 0,C 180,E1 11319.007,E2 11319.007} C_VEL
LIN {X 0,Y 435.594,Z 578.447,A -85,B 0,C 180,E1 11318.851,E2 11318.851} C_VEL
LIN {X 0,Y 413.828,Z 797.611,A -85,B 0,C 180,E1 11315.674,E2 11315.674} C_VEL
LIN {X 0,Y 410.123,Z 822.827,A -85,B 0,C 180,E1 11315.228,E2 11315.228} C_VEL
LIN {X 0,Y 404.683,Z 848.906,A -85,B 0,C 180,E1 11314.623,E2 11314.623} C_VEL
LIN {X 0,Y 399.208,Z 870.053,A -85,B 0,C 180,E1 11314.003,E2 11314.003} C_VEL
LIN {X 0,Y 392.96,Z 890.6,A -85,B 0,C 180,E1 11313.264,E2 11313.264} C_VEL
LIN {X 0,Y 384.29,Z 915.016,A -85,B 0,C 180,E1 11312.205,E2 11312.205} C_VEL
LIN {X 0,Y 374.918,Z 937.373,A -85,B 0,C 180,E1 11311.013,E2 11311.013} C_VEL
LIN {X 0,Y 366.266,Z 955.834,A -85,B 0,C 180,E1 11309.847,E2 11309.847} C_VEL
LIN {X 0,Y 355.9,Z 975.868,A -85,B 0,C 180,E1 11308.347,E2 11308.347} C_VEL
LIN {X 0,Y 343.019,Z 998.052,A -85,B 0,C 180,E1 11306.325,E2 11306.325} C_VEL
LIN {X 0,Y 332.31,Z 1014.829,A -85,B 0,C 180,E1 11304.477,E2 11304.477} C_VEL
LIN {X 0,Y 321.588,Z 1030.426,A -85,B 0,C 180,E1 11302.45,E2 11302.45} C_VEL
LIN {X 0,Y 308.331,Z 1048.407,A -85,B 0,C 180,E1 11299.646,E2 11299.646} C_VEL
LIN {X 0,Y 295.761,Z 1064.051,A -85,B 0,C 180,E1 11296.621,E2 11296.621} C_VEL
LIN {X 0,Y 285.146,Z 1076.639,A -85,B 0,C 180,E1 11293.691,E2 11293.691} C_VEL
LIN {X 0,Y 273.668,Z 1089.715,A -85,B 0,C 180,E1 11290.017,E2 11290.017} C_VEL
LIN {X 0,Y 261.392,Z 1103.106,A -85,B 0,C 180,E1 11285.281,E2 11285.281} C_VEL
LIN {X 0,Y 252.367,Z 1112.79,A -85,B 0,C 180,E1 11281.001,E2 11281.001} C_VEL
LIN {X 0,Y 244.278,Z 1121.569,A -85,B 0,C 180,E1 11276.235,E2 11276.235} C_VEL
LIN {X 0,Y 236.099,Z 1130.759,A -85,B 0,C 180,E1 11269.803,E2 11269.803} C_VEL
LIN {X 0,Y 231.367,Z 1136.556,A -85,B 0,C 180,E1 11264.516,E2 11264.516} C_VEL
LIN {X 0,Y 228.082,Z 1141.204,A -85,B 0,C 180,E1 11259.08,E2 11259.08} C_VEL
LIN {X 0,Y 225.848,Z 1145.307,A -85,B 0,C 180,E1 11252.537,E2 11252.537} C_VEL
LIN {X 0,Y 225.022,Z 1147.561,A -85,B 0,C 180,E1 11246.688,E2 11246.688} C_VEL
LIN {X 0,Y 224.871,Z 1148.646,A -85,B 0,C 180,E1 11241.562,E2 11241.562} C_VEL
LIN {X 0,Y 225.028,Z 1148.899,A -85,B 0,C 180,E1 11236.641,E2 11236.641} C_VEL
LIN {X 0,Y 225.654,Z 1148.328,A -85,B 0,C 180,E1 11231.488,E2 11231.488} C_VEL
LIN {X 0,Y 227.037,Z 1146.899,A -85,B 0,C 180,E1 11226.356,E2 11226.356} C_VEL
LIN {X 0,Y 229.746,Z 1144.35,A -85,B 0,C 180,E1 11220.828,E2 11220.828} C_VEL
LIN {X 0,Y 234.935,Z 1139.937,A -85,B 0,C 180,E1 11214.334,E2 11214.334} C_VEL
LIN {X 0,Y 242.071,Z 1133.942,A -85,B 0,C 180,E1 11208.318,E2 11208.318} C_VEL
LIN {X 0,Y 249.726,Z 1127.739,A -85,B 0,C 180,E1 11203.526,E2 11203.526} C_VEL
LIN {X 0,Y 259.827,Z 1119.564,A -85,B 0,C 180,E1 11198.567,E2 11198.567} C_VEL
LIN {X 0,Y 273.13,Z 1108.403,A -85,B 0,C 180,E1 11193.421,E2 11193.421} C_VEL
LIN {X 0,Y 284.594,Z 1098.392,A -85,B 0,C 180,E1 11189.798,E2 11189.798} C_VEL
LIN {X 0,Y 297.064,Z 1087.022,A -85,B 0,C 180,E1 11186.453,E2 11186.453} C_VEL
LIN {X 0,Y 313.339,Z 1071.161,A -85,B 0,C 180,E1 11182.751,E2 11182.751} C_VEL
LIN {X 0,Y 326.882,Z 1056.87,A -85,B 0,C 180,E1 11180.108,E2 11180.108} C_VEL
LIN {X 0,Y 339.451,Z 1042.676,A -85,B 0,C 180,E1 11177.936,E2 11177.936} C_VEL
LIN {X 0,Y 354.537,Z 1024.272,A -85,B 0,C 180,E1 11175.615,E2 11175.615} C_VEL
LIN {X 0,Y 368.42,Z 1005.353,A -85,B 0,C 180,E1 11173.693,E2 11173.693} C_VEL
LIN {X 0,Y 379.625,Z 988.716,A -85,B 0,C 180,E1 11172.274,E2 11172.274} C_VEL
LIN {X 0,Y 391.419,Z 969.52,A -85,B 0,C 180,E1 11170.897,E2 11170.897} C_VEL
LIN {X 0,Y 404.468,Z 945.439,A -85,B 0,C 180,E1 11169.481,E2 11169.481} C_VEL
LIN {X 0,Y 413.55,Z 926.417,A -85,B 0,C 180,E1 11168.562,E2 11168.562} C_VEL
LIN {X 0,Y 421.799,Z 906.947,A -85,B 0,C 180,E1 11167.756,E2 11167.756} C_VEL
LIN {X 0,Y 430.604,Z 883.097,A -85,B 0,C 180,E1 11166.935,E2 11166.935} C_VEL
LIN {X 0,Y 438.341,Z 857.261,A -85,B 0,C 180,E1 11166.233,E2 11166.233} C_VEL
LIN {X 0,Y 443.383,Z 836.726,A -85,B 0,C 180,E1 11165.785,E2 11165.785} C_VEL
LIN {X 0,Y 447.721,Z 814.567,A -85,B 0,C 180,E1 11165.391,E2 11165.391} C_VEL
LIN {X 0,Y 450.756,Z 793.747,A -85,B 0,C 180,E1 11165.088,E2 11165.088} C_VEL
LIN {X 0,Y 451.57,Z 786.24,A -85,B 0,C 180,E1 11164.856,E2 11164.856} C_VEL
LIN {X 0,Y 452.992,Z 766.73,A -85,B 0,C 180,E1 11163.804,E2 11163.804} C_VEL
LIN {X 0,Y 453.629,Z 760.255,A -85,B 0,C 180,E1 11163.626,E2 11163.626} C_VEL
LIN {X 0,Y 470.327,Z 614.208,A -85,B 0,C 180,E1 11161.706,E2 11161.706} C_VEL
LIN {X 0,Y 469.475,Z 611.802,A -85,B 0,C 180,E1 11157.925,E2 11157.925} C_VEL
LIN {X 0,Y 469.812,Z 613.37,A -85,B 0,C 180,E1 11155.116,E2 11155.116} C_VEL
LIN {X 0,Y 470.536,Z 615.005,A -85,B 0,C 180,E1 11153.347,E2 11153.347} C_VEL
LIN {X 0,Y 448.617,Z 806.869,A -85,B 0,C 180,E1 11150.711,E2 11150.711} C_VEL
LIN {X 0,Y 444.085,Z 834.017,A -85,B 0,C 180,E1 11150.299,E2 11150.299} C_VEL
LIN {X 0,Y 437.864,Z 860.163,A -85,B 0,C 180,E1 11149.851,E2 11149.851} C_VEL
LIN {X 0,Y 431.544,Z 881.8,A -85,B 0,C 180,E1 11149.408,E2 11149.408} C_VEL
LIN {X 0,Y 423.502,Z 905.152,A -85,B 0,C 180,E1 11148.803,E2 11148.803} C_VEL
LIN {X 0,Y 413.017,Z 930.743,A -85,B 0,C 180,E1 11147.968,E2 11147.968} C_VEL
LIN {X 0,Y 403.55,Z 950.938,A -85,B 0,C 180,E1 11147.15,E2 11147.15} C_VEL
LIN {X 0,Y 393.816,Z 969.622,A -85,B 0,C 180,E1 11146.248,E2 11146.248} C_VEL
LIN {X 0,Y 382.746,Z 988.895,A -85,B 0,C 180,E1 11145.141,E2 11145.141} C_VEL
LIN {X 0,Y 367.666,Z 1012.518,A -85,B 0,C 180,E1 11143.479,E2 11143.479} C_VEL
LIN {X 0,Y 354.202,Z 1031.501,A -85,B 0,C 180,E1 11141.819,E2 11141.819} C_VEL
LIN {X 0,Y 341.813,Z 1047.69,A -85,B 0,C 180,E1 11140.126,E2 11140.126} C_VEL
LIN {X 0,Y 328.233,Z 1064.246,A -85,B 0,C 180,E1 11138.058,E2 11138.058} C_VEL
LIN {X 0,Y 311.033,Z 1083.744,A -85,B 0,C 180,E1 11135.03,E2 11135.03} C_VEL
LIN {X 0,Y 297.259,Z 1098.299,A -85,B 0,C 180,E1 11132.205,E2 11132.205} C_VEL
LIN {X 0,Y 284.235,Z 1111.472,A -85,B 0,C 180,E1 11129.096,E2 11129.096} C_VEL
LIN {X 0,Y 271.015,Z 1124.411,A -85,B 0,C 180,E1 11125.358,E2 11125.358} C_VEL
LIN {X 0,Y 255.739,Z 1138.912,A -85,B 0,C 180,E1 11120.023,E2 11120.023} C_VEL
LIN {X 0,Y 245.448,Z 1148.653,A -85,B 0,C 180,E1 11115.47,E2 11115.47} C_VEL
LIN {X 0,Y 236.47,Z 1157.397,A -85,B 0,C 180,E1 11110.437,E2 11110.437} C_VEL
LIN {X 0,Y 227.805,Z 1166.484,A -85,B 0,C 180,E1 11103.877,E2 11103.877} C_VEL
LIN {X 0,Y 221.807,Z 1173.5,A -85,B 0,C 180,E1 11097.084,E2 11097.084} C_VEL
LIN {X 0,Y 218.734,Z 1178.003,A -85,B 0,C 180,E1 11091.45,E2 11091.45} C_VEL
LIN {X 0,Y 217.091,Z 1181.424,A -85,B 0,C 180,E1 11085.768,E2 11085.768} C_VEL
LIN {X 0,Y 216.543,Z 1183.657,A -85,B 0,C 180,E1 11080.411,E2 11080.411} C_VEL
LIN {X 0,Y 216.575,Z 1184.79,A -85,B 0,C 180,E1 11075.83,E2 11075.83} C_VEL
LIN {X 0,Y 216.709,Z 1185.147,A -85,B 0,C 180,E1 11071.058,E2 11071.058} C_VEL
LIN {X 0,Y 216.672,Z 1184.617,A -85,B 0,C 180,E1 11066.296,E2 11066.296} C_VEL
LIN {X 0,Y 216.59,Z 1182.946,A -85,B 0,C 180,E1 11060.97,E2 11060.97} C_VEL
LIN {X 0,Y 216.989,Z 1180.006,A -85,B 0,C 180,E1 11055.319,E2 11055.319} C_VEL
LIN {X 0,Y 218.37,Z 1175.878,A -85,B 0,C 180,E1 11049.636,E2 11049.636} C_VEL
LIN {X 0,Y 220.939,Z 1170.82,A -85,B 0,C 180,E1 11044.238,E2 11044.238} C_VEL
LIN {X 0,Y 224.844,Z 1164.663,A -85,B 0,C 180,E1 11038.947,E2 11038.947} C_VEL
LIN {X 0,Y 230.833,Z 1156.569,A -85,B 0,C 180,E1 11033.291,E2 11033.291} C_VEL
LIN {X 0,Y 240.595,Z 1144.556,A -85,B 0,C 180,E1 11026.709,E2 11026.709} C_VEL
LIN {X 0,Y 249.477,Z 1134.094,A -85,B 0,C 180,E1 11022.146,E2 11022.146} C_VEL
LIN {X 0,Y 259.142,Z 1122.86,A -85,B 0,C 180,E1 11018.085,E2 11018.085} C_VEL
LIN {X 0,Y 271.725,Z 1108.201,A -85,B 0,C 180,E1 11013.737,E2 11013.737} C_VEL
LIN {X 0,Y 285.311,Z 1091.609,A -85,B 0,C 180,E1 11009.845,E2 11009.845} C_VEL
LIN {X 0,Y 296.614,Z 1077.275,A -85,B 0,C 180,E1 11007.071,E2 11007.071} C_VEL
LIN {X 0,Y 308.426,Z 1061.55,A -85,B 0,C 180,E1 11004.517,E2 11004.517} C_VEL
LIN {X 0,Y 322.987,Z 1040.884,A -85,B 0,C 180,E1 11001.768,E2 11001.768} C_VEL
LIN {X 0,Y 335.425,Z 1021.586,A -85,B 0,C 180,E1 10999.685,E2 10999.685} C_VEL
LIN {X 0,Y 346.442,Z 1003.146,A -85,B 0,C 180,E1 10998.018,E2 10998.018} C_VEL
LIN {X 0,Y 358.858,Z 980.536,A -85,B 0,C 180,E1 10996.319,E2 10996.319} C_VEL
LIN {X 0,Y 369.933,Z 957.619,A -85,B 0,C 180,E1 10994.928,E2 10994.928} C_VEL
LIN {X 0,Y 378.613,Z 937.666,A -85,B 0,C 180,E1 10993.918,E2 10993.918} C_VEL
LIN {X 0,Y 386.449,Z 917.529,A -85,B 0,C 180,E1 10993.065,E2 10993.065} C_VEL
LIN {X 0,Y 395.097,Z 892.17,A -85,B 0,C 180,E1 10992.186,E2 10992.186} C_VEL
LIN {X 0,Y 402.206,Z 866.544,A -85,B 0,C 180,E1 10991.501,E2 10991.501} C_VEL
LIN {X 0,Y 407.242,Z 844.543,A -85,B 0,C 180,E1 10991.033,E2 10991.033} C_VEL
LIN {X 0,Y 411.618,Z 819.761,A -85,B 0,C 180,E1 10990.573,E2 10990.573} C_VEL
LIN {X 0,Y 415.755,Z 782.993,A -85,B 0,C 180,E1 10989.999,E2 10989.999} C_VEL
LIN {X 0,Y 434.924,Z 587.714,A -85,B 0,C 180,E1 10987.115,E2 10987.115} C_VEL
LIN {X 0,Y 431.499,Z 580.117,A -85,B 0,C 180,E1 10984.519,E2 10984.519} C_VEL
LIN {X 0,Y 428.91,Z 574.302,A -85,B 0,C 180,E1 10982.071,E2 10982.071} C_VEL
LIN {X 0,Y 427.185,Z 570.738,A -85,B 0,C 180,E1 10980,E2 10980} C_VEL
LIN {X 0,Y 425.697,Z 567.386,A -85,B 0,C 180,E1 10977.442,E2 10977.442} C_VEL
LIN {X 0,Y 424.626,Z 565.236,A -85,B 0,C 180,E1 10973.238,E2 10973.238} C_VEL
LIN {X 0,Y 424.896,Z 566.022,A -85,B 0,C 180,E1 10970.395,E2 10970.395} C_VEL
LIN {X 0,Y 426.014,Z 567.947,A -85,B 0,C 180,E1 10967.599,E2 10967.599} C_VEL
LIN {X 0,Y 427.973,Z 572.232,A -85,B 0,C 180,E1 10964.692,E2 10964.692} C_VEL
LIN {X 0,Y 430.413,Z 577.352,A -85,B 0,C 180,E1 10962.143,E2 10962.143} C_VEL
LIN {X 0,Y 433.226,Z 583.719,A -85,B 0,C 180,E1 10959.807,E2 10959.807} C_VEL
LIN {X 0,Y 411.483,Z 798.524,A -85,B 0,C 180,E1 10956.729,E2 10956.729} C_VEL
LIN {X 0,Y 407.501,Z 824.888,A -85,B 0,C 180,E1 10956.267,E2 10956.267} C_VEL
LIN {X 0,Y 402.053,Z 850.134,A -85,B 0,C 180,E1 10955.683,E2 10955.683} C_VEL
LIN {X 0,Y 396.398,Z 871.499,A -85,B 0,C 180,E1 10955.065,E2 10955.065} C_VEL
LIN {X 0,Y 389.139,Z 894.707,A -85,B 0,C 180,E1 10954.234,E2 10954.234} C_VEL
LIN {X 0,Y 379.929,Z 919.296,A -85,B 0,C 180,E1 10953.144,E2 10953.144} C_VEL
LIN {X 0,Y 371.606,Z 938.665,A -85,B 0,C 180,E1 10952.113,E2 10952.113} C_VEL
LIN {X 0,Y 362.222,Z 958.216,A -85,B 0,C 180,E1 10950.885,E2 10950.885} C_VEL
LIN {X 0,Y 349.964,Z 981.054,A -85,B 0,C 180,E1 10949.152,E2 10949.152} C_VEL
LIN {X 0,Y 338.366,Z 1000.263,A -85,B 0,C 180,E1 10947.369,E2 10947.369} C_VEL
LIN {X 0,Y 327.451,Z 1016.904,A -85,B 0,C 180,E1 10945.531,E2 10945.531} C_VEL
LIN {X 0,Y 314.783,Z 1034.795,A -85,B 0,C 180,E1 10943.172,E2 10943.172} C_VEL
LIN {X 0,Y 301.287,Z 1052.143,A -85,B 0,C 180,E1 10940.347,E2 10940.347} C_VEL
LIN {X 0,Y 289.761,Z 1066.042,A -85,B 0,C 180,E1 10937.598,E2 10937.598} C_VEL
LIN {X 0,Y 278.302,Z 1079.17,A -85,B 0,C 180,E1 10934.473,E2 10934.473} C_VEL
LIN {X 0,Y 264.448,Z 1094.234,A -85,B 0,C 180,E1 10929.998,E2 10929.998} C_VEL
LIN {X 0,Y 254,Z 1105.13,A -85,B 0,C 180,E1 10925.911,E2 10925.911} C_VEL
LIN {X 0,Y 244.753,Z 1114.661,A -85,B 0,C 180,E1 10921.527,E2 10921.527} C_VEL
LIN {X 0,Y 234.797,Z 1125.022,A -85,B 0,C 180,E1 10915.47,E2 10915.47} C_VEL
LIN {X 0,Y 228.105,Z 1132.213,A -85,B 0,C 180,E1 10909.992,E2 10909.992} C_VEL
LIN {X 0,Y 223.479,Z 1137.643,A -85,B 0,C 180,E1 10904.775,E2 10904.775} C_VEL
LIN {X 0,Y 219.867,Z 1142.595,A -85,B 0,C 180,E1 10898.631,E2 10898.631} C_VEL
LIN {X 0,Y 217.718,Z 1146.365,A -85,B 0,C 180,E1 10891.842,E2 10891.842} C_VEL
LIN {X 0,Y 217.019,Z 1148.335,A -85,B 0,C 180,E1 10886.302,E2 10886.302} C_VEL
LIN {X 0,Y 216.894,Z 1149.325,A -85,B 0,C 180,E1 10881.25,E2 10881.25} C_VEL
LIN {X 0,Y 217.071,Z 1149.564,A -85,B 0,C 180,E1 10876.392,E2 10876.392} C_VEL
LIN {X 0,Y 217.758,Z 1149.011,A -85,B 0,C 180,E1 10871.069,E2 10871.069} C_VEL
LIN {X 0,Y 219.262,Z 1147.606,A -85,B 0,C 180,E1 10865.769,E2 10865.769} C_VEL
LIN {X 0,Y 222.031,Z 1145.209,A -85,B 0,C 180,E1 10860.307,E2 10860.307} C_VEL
